KUKA KRL program: MyProgram_078().src

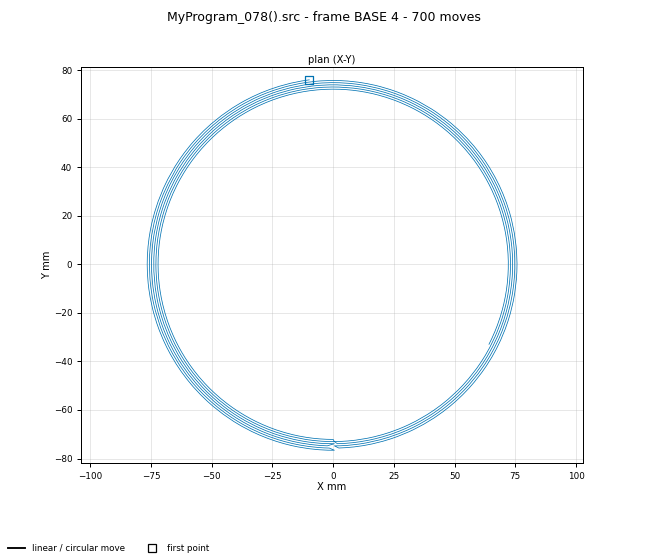
[picture p0: tool path of MyProgram_078().src in frame BASE 4, 700 of 700 moves have a stored position in this frame; points joined in program order, loops and branches not executed]
&ACCESS RVP
&REL 1
&PARAM TEMPLATE = C:\KRC\Roboter\Template\vorgabe
&PARAM EDITMASK = *
DEF MyProgram_078()
; ---- Setting reference (Base) ----
$BASE = BASE_DATA[4]

; --------------------------
; ---- Setting tool (TCP) ----
$TOOL = TOOL_DATA[3]
; --------------------------

$VEL.CP = VEL_APROX_PRINT
Startdeposition()
$VEL.CP = VEL_PRINT
LIN {X -9.8777,Y 75.9494,Z 80,A 92.1088,B 24.884,C -2.486,E1 24.9779,E2 -7.6791} C_DIS
LIN {X -13.075,Y 75.4658,Z 80,A 94.5265,B 24.8842,C -2.4842,E1 24.9713,E2 -10.0948} C_DIS
LIN {X -17.5111,Y 74.5607,Z 80,A 97.8703,B 24.8845,C -2.4802,E1 24.9622,E2 -13.4331} C_DIS
LIN {X -22.3044,Y 73.2687,Z 80,A 101.5575,B 24.885,C -2.4756,E1 24.9523,E2 -17.1153} C_DIS
LIN {X -26.0377,Y 72.0267,Z 80,A 104.8313,B 24.8845,C -2.4806,E1 24.9436,E2 -20.4073} C_DIS
LIN {X -29.6521,Y 70.616,Z 80,A 107.6677,B 24.885,C -2.4749,E1 24.9363,E2 -23.2364} C_DIS
LIN {X -33.18,Y 69.0287,Z 80,A 110.4546,B 24.8857,C -2.4677,E1 24.9292,E2 -26.0132} C_DIS
LIN {X -36.3303,Y 67.4239,Z 80,A 112.8541,B 24.8867,C -2.4571,E1 24.9233,E2 -28.394} C_DIS
LIN {X -38.0419,Y 66.4734,Z 80,A 114.6868,B 24.8861,C -2.4639,E1 24.9188,E2 -30.2484} C_DIS
LIN {X -41.522,Y 64.3565,Z 80,A 117.6505,B 24.8868,C -2.4562,E1 24.9118,E2 -33.2029} C_DIS
LIN {X -46.0253,Y 61.2172,Z 80,A 121.6077,B 24.8879,C -2.4442,E1 24.9029,E2 -37.1451} C_DIS
LIN {X -50.3353,Y 57.7255,Z 80,A 125.8636,B 24.8885,C -2.4378,E1 24.8937,E2 -41.402} C_DIS
LIN {X -53.3197,Y 54.9798,Z 80,A 129.0741,B 24.8887,C -2.4351,E1 24.8872,E2 -44.6194} C_DIS
LIN {X -56.3129,Y 51.9102,Z 80,A 132.6551,B 24.8886,C -2.4366,E1 24.8803,E2 -48.2195} C_DIS
LIN {X -58.7676,Y 49.1151,Z 80,A 135.4497,B 24.8892,C -2.4298,E1 24.8752,E2 -51.0105} C_DIS
LIN {X -61.2757,Y 45.9475,Z 80,A 137.8294,B 24.8914,C -2.4059,E1 24.8713,E2 -53.3446} C_DIS
LIN {X -63.0193,Y 43.5258,Z 80,A 140.4069,B 24.8912,C -2.4083,E1 24.8671,E2 -55.9405} C_DIS
LIN {X -65.1286,Y 40.3019,Z 80,A 143.5889,B 24.8912,C -2.4076,E1 24.8623,E2 -59.1371} C_DIS
LIN {X -68.074,Y 35.0981,Z 80,A 148.6418,B 24.8911,C -2.409,E1 24.8556,E2 -64.22} C_DIS
LIN {X -69.9567,Y 31.1775,Z 80,A 151.3838,B 24.8931,C -2.3867,E1 24.8525,E2 -66.9237} C_DIS
LIN {X -72.0828,Y 25.8816,Z 80,A 155.1336,B 24.8954,C -2.3611,E1 24.8488,E2 -70.6334} C_DIS
LIN {X -73.5664,Y 21.3077,Z 80,A 158.7364,B 24.8964,C -2.3501,E1 24.8458,E2 -74.2305} C_DIS
LIN {X -74.6505,Y 17.1227,Z 80,A 161.6509,B 24.8979,C -2.3323,E1 24.8438,E2 -77.1195} C_DIS
LIN {X -75.2853,Y 14.0748,Z 80,A 164.5038,B 24.8975,C -2.3375,E1 24.8422,E2 -80.0017} C_DIS
LIN {X -75.8096,Y 10.8996,Z 80,A 167.5902,B 24.8967,C -2.3464,E1 24.8409,E2 -83.1278} C_DIS
LIN {X -76.2313,Y 7.3889,Z 80,A 169.9673,B 24.898,C -2.3314,E1 24.8403,E2 -85.4835} C_DIS
LIN {X -76.5241,Y 3.1545,Z 80,A 172.7585,B 24.8997,C -2.312,E1 24.8399,E2 -88.2449} C_DIS
LIN {X -76.5895,Y -0.0837,Z 80,A 175.8098,B 24.8991,C -2.3195,E1 24.8399,E2 -91.3327} C_DIS
LIN {X -76.5051,Y -3.5969,Z 80,A 178.792,B 24.8991,C -2.3199,E1 24.8402,E2 -94.3338} C_DIS
LIN {X -76.1873,Y -7.835,Z 80,A -178.9442,B 24.9018,C -2.2875,E1 24.8408,E2 -96.5338} C_DIS
LIN {X -75.9118,Y -10.1663,Z 80,A -177.0242,B 24.902,C -2.286,E1 24.8415,E2 -98.4617} C_DIS
LIN {X -75.3667,Y -13.6289,Z 80,A -174.4282,B 24.9027,C -2.2773,E1 24.8427,E2 -101.0521} C_DIS
LIN {X -74.423,Y -18.0851,Z 80,A -171.3541,B 24.9043,C -2.2587,E1 24.8446,E2 -104.1} C_DIS
LIN {X -73.9363,Y -19.982,Z 80,A -168.6792,B 24.9021,C -2.284,E1 24.8466,E2 -106.851} C_DIS
LIN {X -72.7026,Y -24.0858,Z 80,A -166.4076,B 24.9049,C -2.2515,E1 24.8485,E2 -109.0578} C_DIS
LIN {X -71.6262,Y -27.1213,Z 80,A -164.2828,B 24.9061,C -2.2375,E1 24.8505,E2 -111.1612} C_DIS
LIN {X -69.8982,Y -31.3073,Z 80,A -160.4907,B 24.9061,C -2.2378,E1 24.8547,E2 -114.9751} C_DIS
LIN {X -68.5056,Y -34.2481,Z 80,A -157.5374,B 24.9055,C -2.244,E1 24.8584,E2 -117.959} C_DIS
LIN {X -66.9906,Y -37.1241,Z 80,A -155.5564,B 24.907,C -2.2262,E1 24.861,E2 -119.9081} C_DIS
LIN {X -64.6632,Y -41.045,Z 80,A -152.4733,B 24.9085,C -2.2091,E1 24.8654,E2 -122.9663} C_DIS
LIN {X -62.5538,Y -44.1917,Z 80,A -149.0219,B 24.9078,C -2.2175,E1 24.8709,E2 -126.4549} C_DIS
LIN {X -59.9723,Y -47.6364,Z 80,A -146.377,B 24.9096,C -2.1954,E1 24.8754,E2 -129.0594} C_DIS
LIN {X -57.6547,Y -50.4164,Z 80,A -143.0708,B 24.9089,C -2.2043,E1 24.8814,E2 -132.4021} C_DIS
LIN {X -54.7215,Y -53.5864,Z 80,A -140.3193,B 24.9104,C -2.1852,E1 24.8866,E2 -135.1198} C_DIS
LIN {X -51.7395,Y -56.4703,Z 80,A -137.0365,B 24.9106,C -2.1835,E1 24.8933,E2 -138.4121} C_DIS
LIN {X -49.3216,Y -58.5956,Z 80,A -134.2933,B 24.9102,C -2.1875,E1 24.8992,E2 -141.1756} C_DIS
LIN {X -45.3584,Y -61.713,Z 80,A -130.7861,B 24.9113,C -2.174,E1 24.9069,E2 -144.6634} C_DIS
LIN {X -40.9195,Y -64.7428,Z 80,A -126.5969,B 24.9115,C -2.1721,E1 24.9167,E2 -148.8618} C_DIS
LIN {X -37.7326,Y -66.6508,Z 80,A -123.7962,B 24.9118,C -2.1688,E1 24.9235,E2 -151.663} C_DIS
LIN {X -33.5371,Y -68.8558,Z 80,A -120.4898,B 24.9126,C -2.1581,E1 24.9317,E2 -154.9528} C_DIS
LIN {X -30.2404,Y -70.3655,Z 80,A -117.2499,B 24.9117,C -2.1693,E1 24.94,E2 -158.2269} C_DIS
LIN {X -26.7617,Y -71.7607,Z 80,A -114.3188,B 24.9117,C -2.1702,E1 24.9477,E2 -161.1663} C_DIS
LIN {X -23.5205,Y -72.888,Z 80,A -112.3294,B 24.9131,C -2.1525,E1 24.9529,E2 -163.1173} C_DIS
LIN {X -20.3575,Y -73.8336,Z 80,A -110.3071,B 24.9142,C -2.1388,E1 24.9582,E2 -165.1103} C_DIS
LIN {X -17.2131,Y -74.6297,Z 80,A -107.234,B 24.9129,C -2.155,E1 24.9667,E2 -168.2263} C_DIS
LIN {X -14.541,Y -75.196,Z 80,A -105.0876,B 24.9127,C -2.1571,E1 24.9726,E2 -170.38} C_DIS
LIN {X -9.9621,Y -75.9385,Z 80,A -101.7452,B 24.9131,C -2.1527,E1 24.9818,E2 -173.7147} C_DIS
LIN {X -5.8541,Y -76.3646,Z 80,A -99.0526,B 24.914,C -2.1415,E1 24.9892,E2 -176.3821} C_DIS
LIN {X -2.2483,Y -76.5559,Z 80,A -96.0072,B 24.9132,C -2.1514,E1 24.9978,E2 -179.4515} C_DIS
LIN {X 0.483,Y -76.5778,Z 80,A -94.1805,B 24.9136,C -2.1459,E1 25.0028,E2 -181.2653} C_DIS
Enddeposition()
LIN {X 0.483,Y -76.5778,Z 80,A -94.1805,B 24.9136,C -2.1459,E1 25.0028,E2 -181.2653} C_DIS
Startdeposition()
$VEL.CP = VEL_PRINT
LIN {X -1.5771,Y -75.6785,Z 80,A -96.5884,B 24.9143,C -2.1375,E1 24.9961,E2 -178.8375} C_DIS
LIN {X -3.5938,Y -75.6104,Z 80,A -98.116,B 24.9143,C -2.1374,E1 24.9918,E2 -177.3091} C_DIS
LIN {X -5.9465,Y -75.4611,Z 80,A -100.5202,B 24.9156,C -2.1208,E1 24.985,E2 -174.8646} C_DIS
LIN {X -10.1334,Y -75.0142,Z 80,A -103.377,B 24.9149,C -2.13,E1 24.9771,E2 -172.0279} C_DIS
LIN {X -13.7763,Y -74.4317,Z 80,A -105.7979,B 24.914,C -2.1407,E1 24.9705,E2 -169.6301} C_DIS
LIN {X -16.8855,Y -73.7877,Z 80,A -109.1458,B 24.9159,C -2.117,E1 24.9612,E2 -166.2216} C_DIS
LIN {X -20.0524,Y -72.9904,Z 80,A -110.7334,B 24.914,C -2.1416,E1 24.9571,E2 -164.69} C_DIS
LIN {X -22.5615,Y -72.2546,Z 80,A -113.5108,B 24.9155,C -2.1222,E1 24.9495,E2 -161.8618} C_DIS
LIN {X -26.4354,Y -70.9282,Z 80,A -116.6648,B 24.9155,C -2.1236,E1 24.9413,E2 -158.7046} C_DIS
LIN {X -29.9531,Y -69.5158,Z 80,A -119.1811,B 24.9145,C -2.1355,E1 24.9348,E2 -156.211} C_DIS
LIN {X -33.8293,Y -67.7146,Z 80,A -122.3374,B 24.914,C -2.1413,E1 24.9269,E2 -153.0603} C_DIS
LIN {X -37.0718,Y -65.9958,Z 80,A -124.7734,B 24.913,C -2.1537,E1 24.921,E2 -150.6469} C_DIS
LIN {X -39.3179,Y -64.6825,Z 80,A -126.8229,B 24.913,C -2.1544,E1 24.9161,E2 -148.593} C_DIS
LIN {X -41.771,Y -63.1263,Z 80,A -129.0307,B 24.9127,C -2.1576,E1 24.9109,E2 -146.3856} C_DIS
LIN {X -44.0945,Y -61.5258,Z 80,A -131.5383,B 24.9132,C -2.1518,E1 24.9051,E2 -143.8555} C_DIS
LIN {X -47.2138,Y -59.1659,Z 80,A -134.6288,B 24.913,C -2.1538,E1 24.8983,E2 -140.7585} C_DIS
LIN {X -50.1177,Y -56.7278,Z 80,A -137.766,B 24.913,C -2.1528,E1 24.8917,E2 -137.6065} C_DIS
LIN {X -53.6914,Y -53.3574,Z 80,A -140.5466,B 24.9106,C -2.1834,E1 24.8862,E2 -134.8874} C_DIS
LIN {X -55.2117,Y -51.7823,Z 80,A -143.3806,B 24.9126,C -2.1583,E1 24.8806,E2 -131.9811} C_DIS
LIN {X -57.7162,Y -48.9745,Z 80,A -145.892,B 24.9114,C -2.1729,E1 24.8761,E2 -129.493} C_DIS
LIN {X -60.2464,Y -45.8274,Z 80,A -148.8534,B 24.9107,C -2.1824,E1 24.8711,E2 -126.5403} C_DIS
LIN {X -63.1999,Y -41.6594,Z 80,A -152.3928,B 24.9092,C -2.1999,E1 24.8655,E2 -123.0252} C_DIS
LIN {X -65.9338,Y -37.1827,Z 80,A -156.1071,B 24.9078,C -2.2164,E1 24.8602,E2 -119.3312} C_DIS
LIN {X -67.8397,Y -33.5776,Z 80,A -159.079,B 24.9069,C -2.2276,E1 24.8564,E2 -116.37} C_DIS
LIN {X -70.1032,Y -28.5527,Z 80,A -163.5729,B 24.9066,C -2.2316,E1 24.8512,E2 -111.8611} C_DIS
LIN {X -71.1408,Y -25.8597,Z 80,A -166.1416,B 24.9068,C -2.2289,E1 24.8487,E2 -109.2714} C_DIS
LIN {X -73.3129,Y -18.84,Z 80,A -171.1553,B 24.9043,C -2.2584,E1 24.8447,E2 -104.2993} C_DIS
LIN {X -74.0337,Y -15.7716,Z 80,A -173.7321,B 24.9041,C -2.2611,E1 24.8431,E2 -101.7139} C_DIS
LIN {X -74.4465,Y -13.6945,Z 80,A -175.7304,B 24.9045,C -2.2568,E1 24.8421,E2 -99.6934} C_DIS
LIN {X -75.1155,Y -9.3522,Z 80,A -178.5608,B 24.9026,C -2.2788,E1 24.8409,E2 -96.8986} C_DIS
LIN {X -75.4572,Y -5.9942,Z 80,A 178.1742,B 24.9033,C -2.2702,E1 24.8401,E2 -93.5936} C_DIS
LIN {X -75.6918,Y 0.7374,Z 80,A 173.3776,B 24.9013,C -2.2934,E1 24.8398,E2 -88.8234} C_DIS
LIN {X -75.5872,Y 4.0345,Z 80,A 170.7099,B 24.901,C -2.2974,E1 24.8401,E2 -86.1493} C_DIS
LIN {X -75.3206,Y 7.5167,Z 80,A 168.0857,B 24.9002,C -2.3063,E1 24.8408,E2 -83.5305} C_DIS
LIN {X -74.7463,Y 11.9525,Z 80,A 165.1359,B 24.8984,C -2.3271,E1 24.8419,E2 -80.6129} C_DIS
LIN {X -73.7542,Y 17.0307,Z 80,A 160.4984,B 24.8988,C -2.3227,E1 24.8446,E2 -75.9375} C_DIS
LIN {X -72.6569,Y 21.2318,Z 80,A 156.66,B 24.899,C -2.3203,E1 24.8475,E2 -72.071} C_DIS
LIN {X -71.4063,Y 25.117,Z 80,A 154.6372,B 24.896,C -2.3544,E1 24.8493,E2 -70.1183} C_DIS
LIN {X -70.0146,Y 28.7687,Z 80,A 151.3832,B 24.8958,C -2.3565,E1 24.8526,E2 -66.851} C_DIS
LIN {X -68.1089,Y 32.9209,Z 80,A 148.5531,B 24.8935,C -2.3823,E1 24.8558,E2 -64.0671} C_DIS
LIN {X -64.5667,Y 39.5085,Z 80,A 142.8168,B 24.8923,C -2.3961,E1 24.8635,E2 -58.3334} C_DIS
LIN {X -62.8936,Y 42.1203,Z 80,A 139.9656,B 24.8927,C -2.3907,E1 24.8678,E2 -55.4549} C_DIS
LIN {X -61.2571,Y 44.4679,Z 80,A 137.5513,B 24.8927,C -2.3907,E1 24.8718,E2 -53.0287} C_DIS
LIN {X -58.5287,Y 48.0021,Z 80,A 134.3381,B 24.8916,C -2.4034,E1 24.8773,E2 -49.8309} C_DIS
LIN {X -55.7959,Y 51.1522,Z 80,A 131.0027,B 24.8913,C -2.4071,E1 24.8835,E2 -46.4893} C_DIS
LIN {X -52.8118,Y 54.2265,Z 80,A 127.5163,B 24.8911,C -2.4091,E1 24.8904,E2 -42.9928} C_DIS
LIN {X -50.1761,Y 56.6759,Z 80,A 124.7811,B 24.8906,C -2.4149,E1 24.8961,E2 -40.2606} C_DIS
LIN {X -46.3964,Y 59.8094,Z 80,A 121.4177,B 24.8891,C -2.4314,E1 24.9034,E2 -36.924} C_DIS
LIN {X -43.5152,Y 61.9371,Z 80,A 119.0724,B 24.8877,C -2.4458,E1 24.9086,E2 -34.6049} C_DIS
LIN {X -39.3079,Y 64.6885,Z 80,A 114.706,B 24.8883,C -2.4392,E1 24.9189,E2 -30.2086} C_DIS
LIN {X -36.5712,Y 66.2751,Z 80,A 112.1957,B 24.8883,C -2.4405,E1 24.925,E2 -27.6941} C_DIS
LIN {X -32.5759,Y 68.3271,Z 80,A 109.1203,B 24.887,C -2.4539,E1 24.9327,E2 -24.6426} C_DIS
LIN {X -29.8634,Y 69.5545,Z 80,A 106.9712,B 24.8864,C -2.4598,E1 24.9381,E2 -22.5024} C_DIS
LIN {X -27.5483,Y 70.5041,Z 80,A 104.5385,B 24.8874,C -2.4489,E1 24.9445,E2 -20.0384} C_DIS
LIN {X -24.5534,Y 71.6031,Z 80,A 102.4647,B 24.8864,C -2.4604,E1 24.9499,E2 -17.9879} C_DIS
LIN {X -20.0121,Y 73.0011,Z 80,A 98.9131,B 24.8859,C -2.4655,E1 24.9594,E2 -14.4425} C_DIS
LIN {X -18.0186,Y 73.5191,Z 80,A 96.4429,B 24.8879,C -2.4439,E1 24.9663,E2 -11.9177} C_DIS
LIN {X -14.0327,Y 74.3834,Z 80,A 94.194,B 24.8857,C -2.4677,E1 24.9723,E2 -9.7227} C_DIS
LIN {X -10.9409,Y 74.9005,Z 80,A 91.886,B 24.8854,C -2.4709,E1 24.9786,E2 -7.4204} C_DIS
LIN {X -7.0765,Y 75.3635,Z 80,A 89.3928,B 24.8842,C -2.4843,E1 24.9855,E2 -4.9575} C_DIS
LIN {X -5.0644,Y 75.5253,Z 80,A 86.3304,B 24.8878,C -2.4453,E1 24.9943,E2 -1.8011} C_DIS
LIN {X -0.5418,Y 75.6931,Z 80,A 83.9367,B 24.8852,C -2.4728,E1 25.0008,E2 0.5272} C_DIS
LIN {X 2.7502,Y 75.6446,Z 80,A 80.8301,B 24.8867,C -2.457,E1 25.0096,E2 3.6708} C_DIS
LIN {X 6.086,Y 75.4495,Z 80,A 78.59,B 24.886,C -2.4645,E1 25.0157,E2 5.8921} C_DIS
LIN {X 10.3575,Y 74.9835,Z 80,A 75.5916,B 24.8854,C -2.4705,E1 25.024,E2 8.8737} C_DIS
LIN {X 13.8407,Y 74.4196,Z 80,A 72.3601,B 24.8869,C -2.4546,E1 25.033,E2 12.1395} C_DIS
LIN {X 17.1405,Y 73.7288,Z 80,A 70.7874,B 24.8846,C -2.4797,E1 25.0371,E2 13.6506} C_DIS
LIN {X 19.3068,Y 73.1924,Z 80,A 68.1739,B 24.887,C -2.4536,E1 25.0443,E2 16.3218} C_DIS
LIN {X 23.3915,Y 71.9901,Z 80,A 64.9215,B 24.8873,C -2.4503,E1 25.053,E2 19.576} C_DIS
LIN {X 26.5408,Y 70.8889,Z 80,A 63.1766,B 24.8856,C -2.4693,E1 25.0574,E2 21.2722} C_DIS
LIN {X 29.0873,Y 69.8825,Z 80,A 60.9184,B 24.8862,C -2.4621,E1 25.0633,E2 23.5423} C_DIS
LIN {X 32.7666,Y 68.2354,Z 80,A 57.806,B 24.8867,C -2.4569,E1 25.0712,E2 26.6592} C_DIS
LIN {X 35.2397,Y 66.9914,Z 80,A 55.4646,B 24.8876,C -2.4474,E1 25.077,E2 29.0166} C_DIS
LIN {X 40.4766,Y 63.9653,Z 80,A 51.5107,B 24.8866,C -2.4582,E1 25.0864,E2 32.9328} C_DIS
LIN {X 42.3299,Y 62.7522,Z 80,A 49.2882,B 24.8882,C -2.4402,E1 25.0917,E2 35.1905} C_DIS
LIN {X 46.4154,Y 59.7947,Z 80,A 45.9821,B 24.8875,C -2.448,E1 25.099,E2 38.4663} C_DIS
LIN {X 48.6468,Y 57.9943,Z 80,A 43.5524,B 24.8886,C -2.4366,E1 25.1043,E2 40.9138} C_DIS
LIN {X 51.5182,Y 55.46,Z 80,A 40.6828,B 24.889,C -2.4317,E1 25.1102,E2 43.7835} C_DIS
LIN {X 55.0143,Y 51.9922,Z 80,A 36.9651,B 24.8897,C -2.4241,E1 25.1175,E2 47.5033} C_DIS
LIN {X 57.9548,Y 48.6943,Z 80,A 33.8949,B 24.8897,C -2.4244,E1 25.1232,E2 50.5588} C_DIS
LIN {X 60.4112,Y 45.6097,Z 80,A 30.3734,B 24.8917,C -2.4018,E1 25.1293,E2 54.1173} C_DIS
LIN {X 62.6825,Y 42.4339,Z 80,A 27.2188,B 24.8929,C -2.3886,E1 25.1343,E2 57.2876} C_DIS
LIN {X 64.457,Y 39.6885,Z 80,A 24.8099,B 24.8933,C -2.384,E1 25.1378,E2 59.695} C_DIS
LIN {X 66.5079,Y 36.1446,Z 80,A 22.251,B 24.8927,C -2.3916,E1 25.1412,E2 62.2227} C_DIS
LIN {X 68.5159,Y 32.1771,Z 80,A 18.8456,B 24.8936,C -2.3811,E1 25.1455,E2 65.6347} C_DIS
LIN {X 69.8894,Y 29.0708,Z 80,A 15.5268,B 24.8962,C -2.3518,E1 25.1491,E2 69.0043} C_DIS
LIN {X 71.3051,Y 25.4018,Z 80,A 13.913,B 24.8934,C -2.3834,E1 25.1506,E2 70.5345} C_DIS
LIN {X 72.6316,Y 21.3171,Z 80,A 10.1653,B 24.8956,C -2.3589,E1 25.1538,E2 74.3188} C_DIS
LIN {X 73.3917,Y 18.5285,Z 80,A 7.457,B 24.8975,C -2.3369,E1 25.1557,E2 77.0636} C_DIS
LIN {X 74.604,Y 12.8095,Z 80,A 3.9207,B 24.8964,C -2.3497,E1 25.1576,E2 80.5489} C_DIS
LIN {X 75.3352,Y 7.3665,Z 80,A -0.1483,B 24.8973,C -2.3394,E1 25.1591,E2 84.6184} C_DIS
LIN {X 75.5228,Y 5.1018,Z 80,A -2.2389,B 24.8988,C -2.3228,E1 25.1595,E2 86.7356} C_DIS
LIN {X 75.694,Y 0.335,Z 80,A -6.1723,B 24.9006,C -2.3017,E1 25.1598,E2 90.6955} C_DIS
LIN {X 75.6309,Y -3.1149,Z 80,A -8.384,B 24.9003,C -2.3054,E1 25.1596,E2 92.8855} C_DIS
LIN {X 75.4373,Y -6.2402,Z 80,A -10.8516,B 24.9012,C -2.2949,E1 25.1591,E2 95.3632} C_DIS
LIN {X 74.7333,Y -12.0356,Z 80,A -14.9146,B 24.9015,C -2.2915,E1 25.1576,E2 99.4102} C_DIS
LIN {X 74.1249,Y -15.3364,Z 80,A -17.626,B 24.9026,C -2.2783,E1 25.1562,E2 102.1368} C_DIS
LIN {X 72.95,Y -20.198,Z 80,A -21.0846,B 24.9028,C -2.2763,E1 25.1539,E2 105.5803} C_DIS
LIN {X 71.9928,Y -23.3813,Z 80,A -24.6347,B 24.9061,C -2.2376,E1 25.1508,E2 109.2016} C_DIS
LIN {X 70.8117,Y -26.7476,Z 80,A -26.1131,B 24.9037,C -2.2658,E1 25.1495,E2 110.605} C_DIS
LIN {X 68.9544,Y -31.2255,Z 80,A -30.6307,B 24.9068,C -2.2293,E1 25.1445,E2 115.184} C_DIS
LIN {X 67.1287,Y -34.9777,Z 80,A -33.3836,B 24.9065,C -2.2321,E1 25.1411,E2 117.9157} C_DIS
LIN {X 65.3574,Y -38.1859,Z 80,A -36.6198,B 24.9083,C -2.2104,E1 25.1365,E2 121.1864} C_DIS
LIN {X 63.124,Y -41.7745,Z 80,A -40.0037,B 24.9095,C -2.1961,E1 25.1314,E2 124.5873} C_DIS
LIN {X 61.155,Y -44.6072,Z 80,A -41.8497,B 24.9083,C -2.2115,E1 25.1284,E2 126.3878} C_DIS
LIN {X 58.0862,Y -48.5361,Z 80,A -45.7317,B 24.9093,C -2.1984,E1 25.1216,E2 130.2827} C_DIS
LIN {X 55.8549,Y -51.0879,Z 80,A -48.965,B 24.9115,C -2.1724,E1 25.1155,E2 133.563} C_DIS
LIN {X 53.3412,Y -53.7074,Z 80,A -50.9656,B 24.9102,C -2.1876,E1 25.1117,E2 135.5193} C_DIS
LIN {X 50.6173,Y -56.2818,Z 80,A -53.7997,B 24.9108,C -2.181,E1 25.1058,E2 138.3573} C_DIS
LIN {X 48.1407,Y -58.4149,Z 80,A -56.5393,B 24.9119,C -2.1678,E1 25.0999,E2 141.1176} C_DIS
LIN {X 45.1335,Y -60.7689,Z 80,A -59.3124,B 24.9121,C -2.1651,E1 25.0938,E2 143.8869} C_DIS
LIN {X 41.5011,Y -63.3042,Z 80,A -62.0188,B 24.9111,C -2.1772,E1 25.0876,E2 146.5557} C_DIS
LIN {X 37.2963,Y -65.8691,Z 80,A -66.1577,B 24.9126,C -2.1585,E1 25.0777,E2 150.7259} C_DIS
LIN {X 32.9711,Y -68.1372,Z 80,A -69.461,B 24.9122,C -2.1636,E1 25.0695,E2 154.008} C_DIS
LIN {X 31.1012,Y -69.0104,Z 80,A -72.6307,B 24.916,C -2.1159,E1 25.0612,E2 157.2829} C_DIS
LIN {X 26.5262,Y -70.8944,Z 80,A -74.8606,B 24.913,C -2.1533,E1 25.0556,E2 159.4193} C_DIS
LIN {X 23.8179,Y -71.8495,Z 80,A -77.9876,B 24.9154,C -2.1238,E1 25.0472,E2 162.6099} C_DIS
LIN {X 20.5212,Y -72.8601,Z 80,A -79.7557,B 24.9138,C -2.1444,E1 25.0426,E2 164.3263} C_DIS
LIN {X 15.9944,Y -73.986,Z 80,A -83.4595,B 24.9144,C -2.1362,E1 25.0325,E2 168.0444} C_DIS
LIN {X 12.3827,Y -74.6753,Z 80,A -86.266,B 24.9146,C -2.1333,E1 25.0247,E2 170.8545} C_DIS
LIN {X 8.6061,Y -75.204,Z 80,A -89.1905,B 24.9149,C -2.1304,E1 25.0166,E2 173.7835} C_DIS
LIN {X 5.4445,Y -75.4989,Z 80,A -91.5056,B 24.9148,C -2.1317,E1 25.0102,E2 176.0944} C_DIS
LIN {X 2.3291,Y -75.6591,Z 80,A -94.7094,B 24.9167,C -2.1081,E1 25.0011,E2 179.3533} C_DIS
LIN {X 2.3291,Y -75.6591,Z 80,A -94.7094,B 24.9167,C -2.1081,E1 25.0011,E2 179.3533} C_DIS
Enddeposition()
LIN {X 0.4812,Y -74.7699,Z 80,A -95.2576,B 24.9136,C -2.1469,E1 24.9998,E2 179.8095} C_DIS
Startdeposition()
$VEL.CP = VEL_PRINT
LIN {X 2.812,Y -74.7476,Z 80,A -92.4237,B 24.9112,C -2.1753,E1 25.0079,E2 176.9086} C_DIS
LIN {X 5.9383,Y -74.5647,Z 80,A -90.0902,B 24.9113,C -2.1746,E1 25.0144,E2 174.5779} C_DIS
LIN {X 10.5837,Y -74.0484,Z 80,A -86.7702,B 24.9117,C -2.1695,E1 25.0236,E2 171.2724} C_DIS
LIN {X 13.6044,Y -73.554,Z 80,A -83.8358,B 24.9102,C -2.1877,E1 25.0318,E2 168.2979} C_DIS
LIN {X 19.3007,Y -72.2683,Z 80,A -79.7389,B 24.9107,C -2.1814,E1 25.0429,E2 164.2217} C_DIS
LIN {X 22.9194,Y -71.2032,Z 80,A -76.547,B 24.9098,C -2.1933,E1 25.0514,E2 161.0074} C_DIS
LIN {X 26.8746,Y -69.8074,Z 80,A -72.7517,B 24.908,C -2.2143,E1 25.0615,E2 157.1706} C_DIS
LIN {X 30.3396,Y -68.3725,Z 80,A -70.6516,B 24.9095,C -2.1963,E1 25.0667,E2 155.1181} C_DIS
LIN {X 33.2038,Y -67.0272,Z 80,A -68.3254,B 24.9095,C -2.1973,E1 25.0725,E2 152.7955} C_DIS
LIN {X 35.4029,Y -65.8928,Z 80,A -66.0422,B 24.9082,C -2.2118,E1 25.0782,E2 150.4847} C_DIS
LIN {X 39.9804,Y -63.2212,Z 80,A -61.7012,B 24.9069,C -2.2275,E1 25.0886,E2 146.1201} C_DIS
LIN {X 42.6642,Y -61.4397,Z 80,A -59.6412,B 24.9075,C -2.2205,E1 25.0933,E2 144.0838} C_DIS
LIN {X 45.9769,Y -59.0017,Z 80,A -56.4694,B 24.9069,C -2.2277,E1 25.1004,E2 140.9063} C_DIS
LIN {X 48.3902,Y -57.0403,Z 80,A -54.4365,B 24.9073,C -2.2227,E1 25.1047,E2 138.8931} C_DIS
LIN {X 51.4102,Y -54.333,Z 80,A -51.2033,B 24.9064,C -2.2336,E1 25.1114,E2 135.6471} C_DIS
LIN {X 54.0361,Y -51.7229,Z 80,A -48.1986,B 24.9054,C -2.2455,E1 25.1173,E2 132.6272} C_DIS
LIN {X 55.8891,Y -49.7155,Z 80,A -46.3181,B 24.9054,C -2.2445,E1 25.1208,E2 130.7575} C_DIS
LIN {X 59.7471,Y -45.0051,Z 80,A -42.0825,B 24.9055,C -2.2439,E1 25.1282,E2 126.5429} C_DIS
LIN {X 62.6709,Y -40.8362,Z 80,A -38.2243,B 24.9047,C -2.2533,E1 25.1343,E2 122.6814} C_DIS
LIN {X 64.4742,Y -37.9246,Z 80,A -34.9338,B 24.9024,C -2.2807,E1 25.1391,E2 119.343} C_DIS
LIN {X 66.2003,Y -34.8232,Z 80,A -32.7037,B 24.903,C -2.2739,E1 25.1421,E2 117.1407} C_DIS
LIN {X 68.0942,Y -30.9583,Z 80,A -29.6504,B 24.9028,C -2.2764,E1 25.1458,E2 114.0979} C_DIS
LIN {X 69.6296,Y -27.3294,Z 80,A -26.6007,B 24.9019,C -2.2864,E1 25.1491,E2 111.0413} C_DIS
LIN {X 71.6282,Y -21.5532,Z 80,A -22.1045,B 24.9012,C -2.2952,E1 25.1531,E2 106.5498} C_DIS
LIN {X 72.9563,Y -16.5124,Z 80,A -17.4227,B 24.8983,C -2.3284,E1 25.1564,E2 101.8164} C_DIS
LIN {X 73.8228,Y -12.0599,Z 80,A -13.4403,B 24.8959,C -2.3549,E1 25.1583,E2 97.7949} C_DIS
LIN {X 74.3269,Y -8.4086,Z 80,A -11.3147,B 24.897,C -2.3426,E1 25.159,E2 95.7107} C_DIS
LIN {X 74.6276,Y -5.0883,Z 80,A -8.8673,B 24.8966,C -2.3476,E1 25.1595,E2 93.2662} C_DIS
LIN {X 74.7805,Y -1.7516,Z 80,A -6.191,B 24.8956,C -2.3593,E1 25.1598,E2 90.5781} C_DIS
LIN {X 74.7622,Y 2.409,Z 80,A -3.4856,B 24.8959,C -2.3549,E1 25.1597,E2 87.8992} C_DIS
LIN {X 74.6559,Y 4.6529,Z 80,A -1.4171,B 24.8945,C -2.3708,E1 25.1593,E2 85.8055} C_DIS
LIN {X 74.3647,Y 8.0611,Z 80,A 1.4492,B 24.8931,C -2.3865,E1 25.1586,E2 82.9191} C_DIS
LIN {X 73.8505,Y 11.8943,Z 80,A 4.7657,B 24.8913,C -2.4064,E1 25.1571,E2 79.5751} C_DIS
LIN {X 73.2334,Y 15.234,Z 80,A 6.7132,B 24.8924,C -2.3946,E1 25.1561,E2 77.6667} C_DIS
LIN {X 72.3845,Y 18.8602,Z 80,A 9.5137,B 24.8918,C -2.4017,E1 25.1542,E2 74.8657} C_DIS
LIN {X 71.1715,Y 23.0171,Z 80,A 13.0341,B 24.8903,C -2.4177,E1 25.1513,E2 71.3275} C_DIS
LIN {X 70.3093,Y 25.5299,Z 80,A 15.355,B 24.889,C -2.4322,E1 25.1491,E2 68.9853} C_DIS
LIN {X 68.6095,Y 29.7973,Z 80,A 18.2292,B 24.8898,C -2.423,E1 25.146,E2 66.1487} C_DIS
LIN {X 67.4211,Y 32.3971,Z 80,A 20.6833,B 24.8885,C -2.437,E1 25.1431,E2 63.6749} C_DIS
LIN {X 65.8164,Y 35.5442,Z 80,A 23.5357,B 24.8875,C -2.4487,E1 25.1393,E2 60.8099} C_DIS
LIN {X 62.8617,Y 40.5415,Z 80,A 27.6478,B 24.8873,C -2.4503,E1 25.1334,E2 56.7148} C_DIS
LIN {X 61.0178,Y 43.2672,Z 80,A 30.3791,B 24.8862,C -2.4628,E1 25.129,E2 53.9673} C_DIS
LIN {X 57.5907,Y 47.7335,Z 80,A 34.5261,B 24.8857,C -2.4681,E1 25.1218,E2 49.8271} C_DIS
LIN {X 55.1061,Y 50.5815,Z 80,A 37.3812,B 24.8852,C -2.4734,E1 25.1165,E2 46.9723} C_DIS
LIN {X 52.2671,Y 53.5111,Z 80,A 40.2054,B 24.8854,C -2.4713,E1 25.111,E2 44.165} C_DIS
LIN {X 50.4341,Y 55.2414,Z 80,A 42.3699,B 24.8844,C -2.482,E1 25.1065,E2 41.9841} C_DIS
LIN {X 47.4522,Y 57.8235,Z 80,A 45.3604,B 24.8839,C -2.4868,E1 25.1002,E2 38.9939} C_DIS
LIN {X 43.9521,Y 60.5252,Z 80,A 49.3052,B 24.8819,C -2.5087,E1 25.0913,E2 35.0113} C_DIS
LIN {X 41.2743,Y 62.3828,Z 80,A 51.1306,B 24.8833,C -2.4936,E1 25.0871,E2 33.2278} C_DIS
LIN {X 38.7436,Y 63.9853,Z 80,A 53.6081,B 24.8825,C -2.5022,E1 25.0812,E2 30.7378} C_DIS
LIN {X 34.533,Y 66.3524,Z 80,A 56.6845,B 24.8836,C -2.4897,E1 25.0738,E2 27.6998} C_DIS
LIN {X 30.9922,Y 68.0786,Z 80,A 60.2601,B 24.8818,C -2.5089,E1 25.0647,E2 24.0883} C_DIS
LIN {X 28.4244,Y 69.1899,Z 80,A 62.2462,B 24.882,C -2.5068,E1 25.0596,E2 22.1118} C_DIS
LIN {X 25.6595,Y 70.2621,Z 80,A 64.8765,B 24.8809,C -2.5188,E1 25.0527,E2 19.4586} C_DIS
LIN {X 22.5779,Y 71.3134,Z 80,A 67.4863,B 24.8804,C -2.5239,E1 25.0457,E2 16.8415} C_DIS
LIN {X 18.6435,Y 72.4403,Z 80,A 70.051,B 24.8817,C -2.5103,E1 25.0389,E2 14.3131} C_DIS
LIN {X 13.4747,Y 73.5776,Z 80,A 74.0849,B 24.8816,C -2.5116,E1 25.0279,E2 10.2813} C_DIS
LIN {X 9.8948,Y 74.1441,Z 80,A 76.9996,B 24.8812,C -2.5161,E1 25.0198,E2 7.3586} C_DIS
LIN {X 6.7902,Y 74.492,Z 80,A 80.3304,B 24.8787,C -2.5416,E1 25.0104,E2 3.9692} C_DIS
LIN {X 2.7304,Y 74.7507,Z 80,A 81.9274,B 24.8826,C -2.501,E1 25.0062,E2 2.4693} C_DIS
LIN {X -0.7522,Y 74.7977,Z 80,A 86.0605,B 24.879,C -2.5392,E1 24.9944,E2 -1.7545} C_DIS
LIN {X -4.6442,Y 74.6565,Z 80,A 87.9785,B 24.8817,C -2.51,E1 24.9893,E2 -3.6037} C_DIS
LIN {X -7.0504,Y 74.4677,Z 80,A 90.2171,B 24.8809,C -2.5193,E1 24.983,E2 -5.8655} C_DIS
LIN {X -12.028,Y 73.8281,Z 80,A 93.5546,B 24.8823,C -2.5038,E1 24.9738,E2 -9.1685} C_DIS
LIN {X -17.5464,Y 72.7132,Z 80,A 98.0526,B 24.8823,C -2.5049,E1 24.9615,E2 -13.6745} C_DIS
LIN {X -22.5224,Y 71.3306,Z 80,A 102.1544,B 24.8823,C -2.5043,E1 24.9505,E2 -17.7817} C_DIS
LIN {X -25.206,Y 70.4255,Z 80,A 104.4085,B 24.8823,C -2.5038,E1 24.9445,E2 -20.0389} C_DIS
LIN {X -30.0757,Y 68.4883,Z 80,A 108.2153,B 24.8833,C -2.493,E1 24.9347,E2 -23.8285} C_DIS
LIN {X -31.9713,Y 67.6247,Z 80,A 110.3235,B 24.8824,C -2.5034,E1 24.9293,E2 -25.9668} C_DIS
LIN {X -36.8142,Y 65.1156,Z 80,A 115.527,B 24.8806,C -2.5222,E1 24.9165,E2 -31.2299} C_DIS
LIN {X -41.2915,Y 62.3715,Z 80,A 118.1988,B 24.8845,C -2.4808,E1 24.9104,E2 -33.8118} C_DIS
LIN {X -43.7699,Y 60.6578,Z 80,A 120.8852,B 24.884,C -2.4855,E1 24.9043,E2 -36.5187} C_DIS
LIN {X -47.1298,Y 58.0858,Z 80,A 123.8792,B 24.8852,C -2.4726,E1 24.8977,E2 -39.4929} C_DIS
LIN {X -49.8558,Y 55.7635,Z 80,A 126.4368,B 24.8862,C -2.462,E1 24.8924,E2 -42.0352} C_DIS
LIN {X -52.6111,Y 53.1715,Z 80,A 129.4619,B 24.8866,C -2.4583,E1 24.8863,E2 -45.064} C_DIS
LIN {X -54.8474,Y 50.8623,Z 80,A 132.0749,B 24.8868,C -2.4559,E1 24.8813,E2 -47.6827} C_DIS
LIN {X -56.8541,Y 48.6087,Z 80,A 134.1595,B 24.8878,C -2.4446,E1 24.8775,E2 -49.7498} C_DIS
LIN {X -58.8273,Y 46.2013,Z 80,A 137.1462,B 24.8871,C -2.4529,E1 24.8722,E2 -52.7702} C_DIS
LIN {X -61.6496,Y 42.3614,Z 80,A 141.0011,B 24.8875,C -2.4479,E1 24.866,E2 -56.6322} C_DIS
LIN {X -63.5056,Y 39.525,Z 80,A 142.6669,B 24.8902,C -2.4184,E1 24.8636,E2 -58.2361} C_DIS
LIN {X -65.7928,Y 35.5878,Z 80,A 146.1256,B 24.8912,C -2.4078,E1 24.8588,E2 -61.6873} C_DIS
LIN {X -67.3861,Y 32.4686,Z 80,A 149.6171,B 24.8902,C -2.419,E1 24.8544,E2 -65.2245} C_DIS
LIN {X -68.9618,Y 28.9728,Z 80,A 152.1017,B 24.892,C -2.3995,E1 24.8517,E2 -67.6763} C_DIS
LIN {X -70.3827,Y 25.3252,Z 80,A 155.0202,B 24.8929,C -2.3885,E1 24.8488,E2 -70.5849} C_DIS
LIN {X -71.7019,Y 21.3076,Z 80,A 157.9073,B 24.8946,C -2.3703,E1 24.8464,E2 -73.4449} C_DIS
LIN {X -72.3095,Y 19.1479,Z 80,A 160.4146,B 24.8934,C -2.3834,E1 24.8445,E2 -75.9981} C_DIS
LIN {X -73.6522,Y 13.0597,Z 80,A 164.6723,B 24.8958,C -2.3562,E1 24.8421,E2 -80.2158} C_DIS
LIN {X -74.0363,Y 10.6684,Z 80,A 166.8589,B 24.8957,C -2.358,E1 24.8412,E2 -82.42} C_DIS
LIN {X -74.4094,Y 7.6447,Z 80,A 169.9649,B 24.8947,C -2.3689,E1 24.8403,E2 -85.5705} C_DIS
LIN {X -74.6993,Y 3.8963,Z 80,A 171.7319,B 24.8978,C -2.3335,E1 24.84,E2 -87.2636} C_DIS
LIN {X -74.7847,Y 1.567,Z 80,A 174.9828,B 24.8953,C -2.3624,E1 24.8398,E2 -90.6032} C_DIS
LIN {X -74.7377,Y -3.077,Z 80,A 178.3131,B 24.8968,C -2.3457,E1 24.8402,E2 -93.9136} C_DIS
LIN {X -74.4727,Y -6.9933,Z 80,A -179.5693,B 24.8994,C -2.3152,E1 24.8407,E2 -95.971} C_DIS
LIN {X -74.1982,Y -9.4773,Z 80,A -177.219,B 24.8991,C -2.3195,E1 24.8415,E2 -98.3457} C_DIS
LIN {X -73.487,Y -13.9596,Z 80,A -174.0912,B 24.9007,C -2.3005,E1 24.8429,E2 -101.4467} C_DIS
LIN {X -72.7573,Y -17.3636,Z 80,A -171.63,B 24.9018,C -2.2875,E1 24.8444,E2 -103.8913} C_DIS
LIN {X -72.1522,Y -19.7295,Z 80,A -168.6267,B 24.9,C -2.3089,E1 24.8467,E2 -106.9631} C_DIS
LIN {X -70.987,Y -23.5784,Z 80,A -166.3654,B 24.9025,C -2.2801,E1 24.8486,E2 -109.1687} C_DIS
LIN {X -69.8409,Y -26.7864,Z 80,A -162.8537,B 24.9012,C -2.2943,E1 24.8522,E2 -112.7339} C_DIS
LIN {X -68.2468,Y -30.6192,Z 80,A -160.6116,B 24.904,C -2.2627,E1 24.8546,E2 -114.9129} C_DIS
LIN {X -67.3815,Y -32.4796,Z 80,A -158.8585,B 24.904,C -2.2627,E1 24.8567,E2 -116.6756} C_DIS
LIN {X -65.6605,Y -35.8317,Z 80,A -156.077,B 24.9048,C -2.2523,E1 24.8603,E2 -119.4472} C_DIS
LIN {X -63.4924,Y -39.5462,Z 80,A -153.1744,B 24.9064,C -2.2343,E1 24.8644,E2 -122.3216} C_DIS
LIN {X -62.2009,Y -41.5492,Z 80,A -149.8361,B 24.9036,C -2.2666,E1 24.8698,E2 -125.7539} C_DIS
LIN {X -59.4863,Y -45.3503,Z 80,A -147.3668,B 24.9067,C -2.2306,E1 24.8738,E2 -128.1491} C_DIS
LIN {X -56.4128,Y -49.1201,Z 80,A -143.2097,B 24.9065,C -2.2327,E1 24.8813,E2 -132.3303} C_DIS
LIN {X -54.0506,Y -51.7084,Z 80,A -140.9106,B 24.9078,C -2.2174,E1 24.8856,E2 -134.6028} C_DIS
LIN {X -49.0215,Y -56.4989,Z 80,A -136.0706,B 24.9096,C -2.1947,E1 24.8954,E2 -139.4086} C_DIS
LIN {X -46.404,Y -58.6672,Z 80,A -132.4286,B 24.9079,C -2.216,E1 24.9034,E2 -143.115} C_DIS
LIN {X -42.642,Y -61.456,Z 80,A -129.3056,B 24.9094,C -2.1982,E1 24.9105,E2 -146.2065} C_DIS
LIN {X -39.8407,Y -63.3084,Z 80,A -126.5622,B 24.9094,C -2.1986,E1 24.9169,E2 -148.9597} C_DIS
LIN {X -37.0046,Y -65.0071,Z 80,A -124.1194,B 24.9098,C -2.1928,E1 24.9228,E2 -151.3959} C_DIS
LIN {X -34.124,Y -66.5637,Z 80,A -121.3393,B 24.9095,C -2.1966,E1 24.9297,E2 -154.1927} C_DIS
LIN {X -29.5386,Y -68.7209,Z 80,A -118.0855,B 24.9112,C -2.1761,E1 24.9379,E2 -157.4057} C_DIS
LIN {X -26.4411,Y -69.9718,Z 80,A -115.4907,B 24.9113,C -2.1745,E1 24.9446,E2 -160.0025} C_DIS
LIN {X -23.3032,Y -71.0779,Z 80,A -112.7172,B 24.911,C -2.1783,E1 24.952,E2 -162.7903} C_DIS
LIN {X -20.6856,Y -71.8843,Z 80,A -110.2462,B 24.9103,C -2.1867,E1 24.9587,E2 -165.2853} C_DIS
LIN {X -16.5579,Y -72.9458,Z 80,A -107.3413,B 24.9112,C -2.1755,E1 24.9665,E2 -168.1674} C_DIS
LIN {X -13.3052,Y -73.6081,Z 80,A -104.7319,B 24.9112,C -2.1763,E1 24.9737,E2 -170.7816} C_DIS
LIN {X -9.2495,Y -74.2272,Z 80,A -100.9193,B 24.9097,C -2.1938,E1 24.9844,E2 -174.6387} C_DIS
LIN {X -5.6937,Y -74.5835,Z 80,A -98.8673,B 24.9113,C -2.1751,E1 24.99,E2 -176.6471} C_DIS
LIN {X -2.4448,Y -74.7611,Z 80,A -95.3893,B 24.909,C -2.2024,E1 24.9998,E2 -180.1905} C_DIS
LIN {X -2.4448,Y -74.7611,Z 80,A -95.3893,B 24.909,C -2.2024,E1 24.9998,E2 -180.1905} C_DIS
Enddeposition()
LIN {X 0.4796,Y -73.8887,Z 80,A -95.0297,B 24.9119,C -2.1674,E1 25.0006,E2 -180.4671} C_DIS
Startdeposition()
$VEL.CP = VEL_PRINT
LIN {X -2.905,Y -73.8495,Z 80,A -97.9552,B 24.9126,C -2.1587,E1 24.9924,E2 -177.5207} C_DIS
LIN {X -5.7008,Y -73.6864,Z 80,A -101.1444,B 24.9147,C -2.1324,E1 24.9833,E2 -174.2677} C_DIS
LIN {X -9.9835,Y -73.2292,Z 80,A -103.4151,B 24.9125,C -2.1605,E1 24.9772,E2 -172.062} C_DIS
LIN {X -12.4125,Y -72.8574,Z 80,A -105.6156,B 24.913,C -2.1534,E1 24.9711,E2 -169.8426} C_DIS
LIN {X -16.2302,Y -72.1034,Z 80,A -108.6426,B 24.913,C -2.1544,E1 24.9628,E2 -166.8145} C_DIS
LIN {X -21.102,Y -70.8303,Z 80,A -113.0879,B 24.9138,C -2.1433,E1 24.9508,E2 -162.3357} C_DIS
LIN {X -24.59,Y -69.6963,Z 80,A -115.2215,B 24.9122,C -2.1634,E1 24.9453,E2 -160.2458} C_DIS
LIN {X -27.9402,Y -68.422,Z 80,A -117.7489,B 24.9115,C -2.1724,E1 24.9387,E2 -157.7342} C_DIS
LIN {X -31.5638,Y -66.8283,Z 80,A -121.6402,B 24.9129,C -2.1554,E1 24.9287,E2 -153.7929} C_DIS
LIN {X -35.9019,Y -64.6011,Z 80,A -124.7513,B 24.9111,C -2.1767,E1 24.9212,E2 -150.7239} C_DIS
LIN {X -38.3119,Y -63.2015,Z 80,A -126.9465,B 24.9109,C -2.179,E1 24.9159,E2 -148.5274} C_DIS
LIN {X -41.0409,Y -61.4652,Z 80,A -129.5533,B 24.9109,C -2.1804,E1 24.9098,E2 -145.9156} C_DIS
LIN {X -43.9772,Y -59.4,Z 80,A -133.2227,B 24.9122,C -2.1638,E1 24.9014,E2 -142.1936} C_DIS
LIN {X -47.1639,Y -56.9016,Z 80,A -135.4526,B 24.9099,C -2.1913,E1 24.8967,E2 -140.0208} C_DIS
LIN {X -49.3949,Y -54.9762,Z 80,A -138.5264,B 24.9111,C -2.1769,E1 24.8902,E2 -136.9007} C_DIS
LIN {X -52.082,Y -52.4378,Z 80,A -140.6737,B 24.9092,C -2.1999,E1 24.886,E2 -134.799} C_DIS
LIN {X -53.9137,Y -50.5524,Z 80,A -143.5696,B 24.9105,C -2.1841,E1 24.8804,E2 -131.8527} C_DIS
LIN {X -56.596,Y -47.5317,Z 80,A -145.5779,B 24.9078,C -2.2175,E1 24.8769,E2 -129.9151} C_DIS
LIN {X -58.1096,Y -45.6676,Z 80,A -147.6916,B 24.9078,C -2.216,E1 24.8732,E2 -127.7877} C_DIS
LIN {X -59.3828,Y -44.0006,Z 80,A -149.9231,B 24.9087,C -2.2057,E1 24.8694,E2 -125.5211} C_DIS
LIN {X -62.0663,Y -40.1255,Z 80,A -152.9598,B 24.9068,C -2.2293,E1 24.8647,E2 -122.5255} C_DIS
LIN {X -63.7785,Y -37.3445,Z 80,A -155.8874,B 24.907,C -2.2267,E1 24.8605,E2 -119.5766} C_DIS
LIN {X -66.3179,Y -32.6204,Z 80,A -159.4524,B 24.9049,C -2.2517,E1 24.856,E2 -116.0524} C_DIS
LIN {X -67.9256,Y -29.1251,Z 80,A -163.2981,B 24.9058,C -2.2403,E1 24.8515,E2 -112.1582} C_DIS
LIN {X -69.6798,Y -24.6368,Z 80,A -166.4337,B 24.9038,C -2.2648,E1 24.8485,E2 -109.0635} C_DIS
LIN {X -70.9598,Y -20.6656,Z 80,A -169.8567,B 24.9033,C -2.2701,E1 24.8457,E2 -105.6334} C_DIS
LIN {X -71.8725,Y -17.219,Z 80,A -172.1699,B 24.9017,C -2.2888,E1 24.8441,E2 -103.3513} C_DIS
LIN {X -72.5141,Y -14.2823,Z 80,A -175.4648,B 24.903,C -2.274,E1 24.8422,E2 -100.0017} C_DIS
LIN {X -73.2747,Y -9.6471,Z 80,A -178.6269,B 24.9011,C -2.2962,E1 24.8409,E2 -96.8736} C_DIS
LIN {X -73.8469,Y -2.9745,Z 80,A 176.553,B 24.8989,C -2.321,E1 24.8399,E2 -92.0838} C_DIS
LIN {X -73.8647,Y 2.4986,Z 80,A 172.2044,B 24.898,C -2.332,E1 24.8399,E2 -87.7354} C_DIS
LIN {X -73.5999,Y 6.7289,Z 80,A 168.7173,B 24.8974,C -2.3379,E1 24.8406,E2 -84.2414} C_DIS
LIN {X -73.2642,Y 9.7277,Z 80,A 166.266,B 24.897,C -2.3428,E1 24.8414,E2 -81.7872} C_DIS
LIN {X -72.7944,Y 12.778,Z 80,A 163.9022,B 24.8963,C -2.351,E1 24.8425,E2 -79.4289} C_DIS
LIN {X -71.9615,Y 16.8467,Z 80,A 160.4904,B 24.8958,C -2.3568,E1 24.8445,E2 -76.0109} C_DIS
LIN {X -70.9862,Y 20.5751,Z 80,A 157.882,B 24.8942,C -2.3747,E1 24.8464,E2 -73.43} C_DIS
LIN {X -70.22,Y 23.0497,Z 80,A 155.7798,B 24.8938,C -2.3788,E1 24.8482,E2 -71.3255} C_DIS
LIN {X -69.4781,Y 25.1993,Z 80,A 153.6766,B 24.894,C -2.3764,E1 24.8501,E2 -69.2048} C_DIS
LIN {X -67.8878,Y 29.2127,Z 80,A 150.0062,B 24.8938,C -2.3792,E1 24.8541,E2 -65.5207} C_DIS
LIN {X -65.3889,Y 34.4454,Z 80,A 145.9417,B 24.8917,C -2.4022,E1 24.8591,E2 -61.4891} C_DIS
LIN {X -63.3071,Y 38.1381,Z 80,A 142.8246,B 24.8905,C -2.4154,E1 24.8634,E2 -58.3874} C_DIS
LIN {X -60.3911,Y 42.6052,Z 80,A 138.7716,B 24.8893,C -2.4287,E1 24.8696,E2 -54.3458} C_DIS
LIN {X -59.138,Y 44.3274,Z 80,A 136.5379,B 24.8901,C -2.4197,E1 24.8734,E2 -52.0799} C_DIS
LIN {X -56.6543,Y 47.4615,Z 80,A 133.8219,B 24.8886,C -2.4366,E1 24.8781,E2 -49.3915} C_DIS
LIN {X -54.6739,Y 49.7288,Z 80,A 131.0555,B 24.889,C -2.4324,E1 24.8833,E2 -46.6028} C_DIS
LIN {X -51.0941,Y 53.4009,Z 80,A 127.2985,B 24.8876,C -2.447,E1 24.8907,E2 -42.8646} C_DIS
LIN {X -49.2082,Y 55.1433,Z 80,A 124.7255,B 24.8885,C -2.4379,E1 24.8961,E2 -40.2598} C_DIS
LIN {X -46.7706,Y 57.2254,Z 80,A 122.6587,B 24.8871,C -2.4531,E1 24.9005,E2 -38.2212} C_DIS
LIN {X -44.0281,Y 59.3613,Z 80,A 120.0313,B 24.8864,C -2.4602,E1 24.9063,E2 -35.6015} C_DIS
LIN {X -41.3187,Y 61.2781,Z 80,A 117.8045,B 24.8852,C -2.4735,E1 24.9114,E2 -33.3987} C_DIS
LIN {X -37.5076,Y 63.6821,Z 80,A 114.3459,B 24.8845,C -2.4808,E1 24.9196,E2 -29.9466} C_DIS
LIN {X -35.784,Y 64.6668,Z 80,A 112.438,B 24.8851,C -2.4746,E1 24.9242,E2 -28.0183} C_DIS
LIN {X -31.3657,Y 66.9212,Z 80,A 108.7541,B 24.8841,C -2.4846,E1 24.9334,E2 -24.3485} C_DIS
LIN {X -28.2407,Y 68.298,Z 80,A 105.9994,B 24.8841,C -2.4858,E1 24.9405,E2 -21.5902} C_DIS
LIN {X -25.3656,Y 69.4176,Z 80,A 103.5652,B 24.8838,C -2.4879,E1 24.9468,E2 -19.1559} C_DIS
LIN {X -22.2751,Y 70.4712,Z 80,A 100.5838,B 24.8846,C -2.4798,E1 24.9548,E2 -16.1499} C_DIS
LIN {X -18.0375,Y 71.6715,Z 80,A 96.9886,B 24.8846,C -2.4788,E1 24.9646,E2 -12.547} C_DIS
LIN {X -14.8526,Y 72.3987,Z 80,A 95.0572,B 24.8831,C -2.4958,E1 24.9697,E2 -10.6537} C_DIS
LIN {X -8.6997,Y 73.3928,Z 80,A 90.2556,B 24.8827,C -2.4998,E1 24.983,E2 -5.8574} C_DIS
LIN {X -5.8677,Y 73.6735,Z 80,A 88.0801,B 24.8825,C -2.5016,E1 24.989,E2 -3.6852} C_DIS
LIN {X -1.5662,Y 73.8905,Z 80,A 84.681,B 24.8825,C -2.5011,E1 24.9985,E2 -0.2843} C_DIS
LIN {X 1.6141,Y 73.8896,Z 80,A 82.4231,B 24.882,C -2.5069,E1 25.0048,E2 1.9598} C_DIS
LIN {X 7.5013,Y 73.525,Z 80,A 77.6951,B 24.8824,C -2.5027,E1 25.018,E2 6.6954} C_DIS
LIN {X 12.7408,Y 72.801,Z 80,A 73.8918,B 24.8818,C -2.5094,E1 25.0284,E2 10.4795} C_DIS
LIN {X 17.626,Y 71.7743,Z 80,A 68.7828,B 24.885,C -2.475,E1 25.0425,E2 15.6632} C_DIS
LIN {X 21.4722,Y 70.7184,Z 80,A 66.6398,B 24.8829,C -2.4978,E1 25.0481,E2 17.7485} C_DIS
LIN {X 25.121,Y 69.5062,Z 80,A 63.6613,B 24.8831,C -2.4953,E1 25.056,E2 20.7269} C_DIS
LIN {X 28.1489,Y 68.3362,Z 80,A 61.1851,B 24.8833,C -2.4939,E1 25.0624,E2 23.201} C_DIS
LIN {X 31.2783,Y 66.9613,Z 80,A 58.664,B 24.8833,C -2.4944,E1 25.0688,E2 25.7146} C_DIS
LIN {X 33.6174,Y 65.8186,Z 80,A 55.8331,B 24.8855,C -2.4699,E1 25.076,E2 28.5958} C_DIS
LIN {X 36.5087,Y 64.2609,Z 80,A 53.8991,B 24.8843,C -2.483,E1 25.0806,E2 30.4931} C_DIS
LIN {X 39.0502,Y 62.748,Z 80,A 51.6667,B 24.8844,C -2.4812,E1 25.0859,E2 32.7228} C_DIS
LIN {X 41.1156,Y 61.4156,Z 80,A 49.2575,B 24.886,C -2.4644,E1 25.0916,E2 35.1638} C_DIS
LIN {X 45.9736,Y 57.8678,Z 80,A 44.5092,B 24.887,C -2.4539,E1 25.1022,E2 39.9197} C_DIS
LIN {X 49.5843,Y 54.8058,Z 80,A 41.4402,B 24.8861,C -2.4634,E1 25.1086,E2 42.954} C_DIS
LIN {X 51.6336,Y 52.8801,Z 80,A 39.2436,B 24.8866,C -2.4585,E1 25.113,E2 45.1533} C_DIS
LIN {X 54.6163,Y 49.793,Z 80,A 35.4651,B 24.8884,C -2.4386,E1 25.1203,E2 48.9622} C_DIS
LIN {X 57.0856,Y 46.9414,Z 80,A 32.2421,B 24.8898,C -2.4235,E1 25.126,E2 52.2062} C_DIS
LIN {X 59.3976,Y 43.9806,Z 80,A 30.1184,B 24.8884,C -2.4387,E1 25.1295,E2 54.2838} C_DIS
LIN {X 61.2333,Y 41.3848,Z 80,A 27.6682,B 24.8889,C -2.4329,E1 25.1334,E2 56.7356} C_DIS
LIN {X 62.9607,Y 38.708,Z 80,A 25.5191,B 24.8887,C -2.4357,E1 25.1366,E2 58.8672} C_DIS
LIN {X 65.0299,Y 35.1191,Z 80,A 22.1586,B 24.8898,C -2.4229,E1 25.1413,E2 62.2407} C_DIS
LIN {X 66.4563,Y 32.339,Z 80,A 19.6114,B 24.8908,C -2.4126,E1 25.1445,E2 64.7985} C_DIS
LIN {X 67.6376,Y 29.7899,Z 80,A 17.3994,B 24.8914,C -2.4055,E1 25.147,E2 67.0152} C_DIS
LIN {X 68.5268,Y 27.6828,Z 80,A 15.4659,B 24.8923,C -2.3958,E1 25.1491,E2 68.961} C_DIS
LIN {X 69.6155,Y 24.8162,Z 80,A 12.3855,B 24.8947,C -2.3687,E1 25.152,E2 72.0882} C_DIS
LIN {X 70.9166,Y 20.8112,Z 80,A 10.0595,B 24.8932,C -2.386,E1 25.1538,E2 74.3602} C_DIS
LIN {X 71.9474,Y 16.9014,Z 80,A 6.8696,B 24.8942,C -2.3749,E1 25.156,E2 77.5579} C_DIS
LIN {X 72.6842,Y 13.3837,Z 80,A 3.8943,B 24.8954,C -2.3608,E1 25.1576,E2 80.5491} C_DIS
LIN {X 73.1891,Y 10.276,Z 80,A 1.7872,B 24.8952,C -2.3629,E1 25.1585,E2 82.6387} C_DIS
LIN {X 73.578,Y 6.9627,Z 80,A -0.7914,B 24.8959,C -2.355,E1 25.1592,E2 85.2207} C_DIS
LIN {X 73.8044,Y 3.8877,Z 80,A -3.1536,B 24.8965,C -2.3483,E1 25.1596,E2 87.5848} C_DIS
LIN {X 73.8912,Y 1.5285,Z 80,A -4.9262,B 24.8969,C -2.3442,E1 25.1598,E2 89.3567} C_DIS
LIN {X 73.8873,Y -1.7088,Z 80,A -7.5014,B 24.8978,C -2.3343,E1 25.1597,E2 91.9398} C_DIS
LIN {X 73.7405,Y -4.9553,Z 80,A -9.9939,B 24.8984,C -2.327,E1 25.1593,E2 94.4347} C_DIS
LIN {X 73.4477,Y -8.2258,Z 80,A -12.3613,B 24.8987,C -2.3241,E1 25.1587,E2 96.7949} C_DIS
LIN {X 72.9334,Y -11.9577,Z 80,A -15.3723,B 24.8997,C -2.3122,E1 25.1574,E2 99.8163} C_DIS
LIN {X 72.102,Y -16.2365,Z 80,A -18.8216,B 24.9008,C -2.2995,E1 25.1555,E2 103.2756} C_DIS
LIN {X 71.3172,Y -19.3932,Z 80,A -21.3039,B 24.9014,C -2.2927,E1 25.1537,E2 105.7596} C_DIS
LIN {X 70.2565,Y -22.9404,Z 80,A -24.916,B 24.904,C -2.2623,E1 25.1506,E2 109.423} C_DIS
LIN {X 68.9733,Y -26.5527,Z 80,A -26.8994,B 24.9023,C -2.2819,E1 25.1487,E2 111.349} C_DIS
LIN {X 67.6222,Y -29.8248,Z 80,A -29.4773,B 24.9026,C -2.2785,E1 25.146,E2 113.9208} C_DIS
LIN {X 65.6172,Y -34.0082,Z 80,A -33.2739,B 24.904,C -2.262,E1 25.1413,E2 117.736} C_DIS
LIN {X 63.376,Y -38.0242,Z 80,A -36.9451,B 24.9051,C -2.2487,E1 25.1362,E2 121.4196} C_DIS
LIN {X 61.5779,Y -40.8709,Z 80,A -40.4538,B 24.9079,C -2.2156,E1 25.1307,E2 124.989} C_DIS
LIN {X 59.1552,Y -44.3046,Z 80,A -44.0098,B 24.9093,C -2.1984,E1 25.1247,E2 128.5687} C_DIS
LIN {X 55.9639,Y -48.2734,Z 80,A -46.3538,B 24.9064,C -2.234,E1 25.1207,E2 130.8179} C_DIS
LIN {X 53.6535,Y -50.8275,Z 80,A -49.528,B 24.9081,C -2.2128,E1 25.1146,E2 134.028} C_DIS
LIN {X 50.5879,Y -53.8798,Z 80,A -53.1673,B 24.9095,C -2.1968,E1 25.1072,E2 137.6902} C_DIS
LIN {X 47.7523,Y -56.4092,Z 80,A -55.9114,B 24.9095,C -2.1959,E1 25.1014,E2 140.4258} C_DIS
LIN {X 43.9529,Y -59.4179,Z 80,A -59.0157,B 24.9087,C -2.2063,E1 25.0947,E2 143.4939} C_DIS
LIN {X 41.395,Y -61.2264,Z 80,A -61.7393,B 24.9098,C -2.1931,E1 25.0884,E2 146.2393} C_DIS
LIN {X 39.4522,Y -62.4969,Z 80,A -63.6583,B 24.9103,C -2.1864,E1 25.0838,E2 148.1682} C_DIS
LIN {X 36.365,Y -64.3424,Z 80,A -66.3906,B 24.9106,C -2.1829,E1 25.0772,E2 150.9004} C_DIS
LIN {X 33.438,Y -65.9103,Z 80,A -68.9383,B 24.9109,C -2.1794,E1 25.0709,E2 153.4494} C_DIS
LIN {X 30.2491,Y -67.4331,Z 80,A -71.2438,B 24.9103,C -2.1872,E1 25.0652,E2 155.7305} C_DIS
LIN {X 27.2669,Y -68.6935,Z 80,A -73.7217,B 24.9105,C -2.1844,E1 25.0588,E2 158.2091} C_DIS
LIN {X 24.0339,Y -69.8912,Z 80,A -76.9566,B 24.912,C -2.1655,E1 25.0502,E2 161.4822} C_DIS
LIN {X 20.4357,Y -71.0259,Z 80,A -79.7548,B 24.912,C -2.1656,E1 25.0427,E2 164.2751} C_DIS
LIN {X 17.2139,Y -71.8737,Z 80,A -82.2831,B 24.9121,C -2.1645,E1 25.0359,E2 166.8022} C_DIS
LIN {X 14.8664,Y -72.3959,Z 80,A -84.9432,B 24.914,C -2.1416,E1 25.0285,E2 169.5135} C_DIS
LIN {X 11.1013,Y -73.0686,Z 80,A -86.7095,B 24.9116,C -2.1715,E1 25.0238,E2 171.2071} C_DIS
LIN {X 8.1934,Y -73.4512,Z 80,A -89.3607,B 24.9125,C -2.1599,E1 25.0164,E2 173.8837} C_DIS
LIN {X 5.0638,Y -73.7332,Z 80,A -91.8162,B 24.9126,C -2.1582,E1 25.0095,E2 176.3419} C_DIS
LIN {X 1.7403,Y -73.8864,Z 80,A -94.97,B 24.9139,C -2.1422,E1 25.0006,E2 179.5329} C_DIS
LIN {X 1.7403,Y -73.8864,Z 80,A -94.97,B 24.9139,C -2.1422,E1 25.0006,E2 179.5329} C_DIS
Enddeposition()
LIN {X 0.4724,Y -73.0059,Z 80,A -94.7223,B 24.91,C -2.1901,E1 25.0016,E2 179.1716} C_DIS
Startdeposition()
$VEL.CP = VEL_PRINT
LIN {X 3.1492,Y -72.9448,Z 80,A -92.1368,B 24.9089,C -2.2035,E1 25.0089,E2 176.5548} C_DIS
LIN {X 6.0764,Y -72.7597,Z 80,A -89.8459,B 24.9089,C -2.2043,E1 25.0153,E2 174.2632} C_DIS
LIN {X 9.1865,Y -72.4328,Z 80,A -87.3594,B 24.9087,C -2.2067,E1 25.0222,E2 171.7729} C_DIS
LIN {X 14.0285,Y -71.6528,Z 80,A -83.5844,B 24.9086,C -2.2076,E1 25.0326,E2 167.9997} C_DIS
LIN {X 16.8822,Y -71.0339,Z 80,A -81.2266,B 24.9083,C -2.2115,E1 25.039,E2 165.6358} C_DIS
LIN {X 20.3405,Y -70.1234,Z 80,A -78.4219,B 24.908,C -2.2145,E1 25.0466,E2 162.8287} C_DIS
LIN {X 23.2857,Y -69.2,Z 80,A -76.103,B 24.908,C -2.2145,E1 25.0527,E2 160.514} C_DIS
LIN {X 26.9321,Y -67.8644,Z 80,A -73.2697,B 24.9082,C -2.2127,E1 25.0601,E2 157.6911} C_DIS
LIN {X 29.0584,Y -66.9808,Z 80,A -71.5622,B 24.9082,C -2.2125,E1 25.0645,E2 155.988} C_DIS
LIN {X 31.0894,Y -66.0636,Z 80,A -69.3727,B 24.9069,C -2.2275,E1 25.0701,E2 153.7686} C_DIS
LIN {X 34.2073,Y -64.504,Z 80,A -66.7563,B 24.9069,C -2.2287,E1 25.0766,E2 151.1566} C_DIS
LIN {X 38.87,Y -61.8064,Z 80,A -62.4722,B 24.906,C -2.238,E1 25.0869,E2 146.8637} C_DIS
LIN {X 41.6739,Y -59.9512,Z 80,A -59.8483,B 24.9056,C -2.2428,E1 25.093,E2 144.2374} C_DIS
LIN {X 44.5958,Y -57.8107,Z 80,A -56.3951,B 24.9036,C -2.2663,E1 25.1007,E2 140.7411} C_DIS
LIN {X 47.2298,Y -55.6798,Z 80,A -54.4052,B 24.9048,C -2.2529,E1 25.1049,E2 138.7906} C_DIS
LIN {X 51.409,Y -51.8459,Z 80,A -50.5781,B 24.9054,C -2.2454,E1 25.1127,E2 134.9967} C_DIS
LIN {X 53.2697,Y -49.9321,Z 80,A -47.5941,B 24.9028,C -2.2761,E1 25.1186,E2 131.953} C_DIS
LIN {X 55.8592,Y -47.019,Z 80,A -44.3256,B 24.9016,C -2.29,E1 25.1245,E2 128.6664} C_DIS
LIN {X 59.0658,Y -42.9205,Z 80,A -40.5983,B 24.9016,C -2.2905,E1 25.1308,E2 124.9557} C_DIS
LIN {X 60.9422,Y -40.2108,Z 80,A -38.2586,B 24.9016,C -2.2905,E1 25.1344,E2 122.6278} C_DIS
LIN {X 62.6542,Y -37.4887,Z 80,A -35.6909,B 24.9008,C -2.2989,E1 25.1382,E2 120.0532} C_DIS
LIN {X 64.4875,Y -34.2387,Z 80,A -31.5777,B 24.897,C -2.3425,E1 25.1437,E2 115.8587} C_DIS
LIN {X 66.6526,Y -29.805,Z 80,A -29.3962,B 24.9004,C -2.304,E1 25.1461,E2 113.7799} C_DIS
LIN {X 67.5056,Y -27.8177,Z 80,A -27.3327,B 24.899,C -2.3199,E1 25.1484,E2 111.6902} C_DIS
LIN {X 68.816,Y -24.397,Z 80,A -24.8697,B 24.8993,C -2.3166,E1 25.1508,E2 109.2487} C_DIS
LIN {X 69.5886,Y -22.1008,Z 80,A -22.4927,B 24.8976,C -2.3364,E1 25.1529,E2 106.8383} C_DIS
LIN {X 70.4776,Y -19.0729,Z 80,A -20.0697,B 24.897,C -2.3426,E1 25.1547,E2 104.4146} C_DIS
LIN {X 71.2163,Y -16.1005,Z 80,A -17.6985,B 24.8965,C -2.3492,E1 25.1562,E2 102.0416} C_DIS
LIN {X 71.9499,Y -12.4186,Z 80,A -15.0547,B 24.8965,C -2.3496,E1 25.1576,E2 99.4123} C_DIS
LIN {X 72.2617,Y -10.446,Z 80,A -13.0671,B 24.8949,C -2.367,E1 25.1584,E2 97.3954} C_DIS
LIN {X 72.667,Y -7.0926,Z 80,A -10.5937,B 24.8946,C -2.3702,E1 25.1592,E2 94.929} C_DIS
LIN {X 72.9072,Y -3.9208,Z 80,A -8.1209,B 24.8939,C -2.3774,E1 25.1596,E2 92.4537} C_DIS
LIN {X 73.0094,Y -0.7704,Z 80,A -5.6798,B 24.8933,C -2.3843,E1 25.1598,E2 90.0109} C_DIS
LIN {X 72.9955,Y 1.6059,Z 80,A -3.806,B 24.8928,C -2.3905,E1 25.1597,E2 88.1335} C_DIS
LIN {X 72.8801,Y 4.4049,Z 80,A -1.5594,B 24.892,C -2.3989,E1 25.1594,E2 85.8805} C_DIS
LIN {X 72.618,Y 7.582,Z 80,A 0.9986,B 24.8911,C -2.4084,E1 25.1587,E2 83.3152} C_DIS
LIN {X 72.2805,Y 10.315,Z 80,A 3.3585,B 24.89,C -2.421,E1 25.1578,E2 80.9394} C_DIS
LIN {X 71.5018,Y 14.7775,Z 80,A 6.3506,B 24.8905,C -2.4154,E1 25.1563,E2 77.978} C_DIS
LIN {X 71.0144,Y 16.963,Z 80,A 8.3218,B 24.8894,C -2.4271,E1 25.155,E2 75.9908} C_DIS
LIN {X 70.0368,Y 20.6332,Z 80,A 12.2076,B 24.8862,C -2.4627,E1 25.1519,E2 72.0432} C_DIS
LIN {X 68.759,Y 24.5559,Z 80,A 14.3718,B 24.8882,C -2.4406,E1 25.15,E2 69.9431} C_DIS
LIN {X 67.6754,Y 27.4031,Z 80,A 16.8594,B 24.8873,C -2.4503,E1 25.1475,E2 67.4465} C_DIS
LIN {X 66.4735,Y 30.2024,Z 80,A 19.2235,B 24.8868,C -2.4563,E1 25.1448,E2 65.0812} C_DIS
LIN {X 65.1179,Y 33.024,Z 80,A 21.7287,B 24.886,C -2.4645,E1 25.1417,E2 62.5699} C_DIS
LIN {X 63.3811,Y 36.2453,Z 80,A 24.3264,B 24.886,C -2.4643,E1 25.1382,E2 59.9863} C_DIS
LIN {X 62.06,Y 38.4641,Z 80,A 26.4652,B 24.8852,C -2.4728,E1 25.1351,E2 57.8383} C_DIS
LIN {X 60.5989,Y 40.7272,Z 80,A 28.5714,B 24.8848,C -2.4779,E1 25.1319,E2 55.7304} C_DIS
LIN {X 58.8755,Y 43.1804,Z 80,A 30.9793,B 24.8841,C -2.4853,E1 25.1279,E2 53.3168} C_DIS
LIN {X 56.3206,Y 46.4642,Z 80,A 34.2287,B 24.8834,C -2.4926,E1 25.1223,E2 50.0654} C_DIS
LIN {X 54.2186,Y 48.9006,Z 80,A 37.5903,B 24.8806,C -2.5221,E1 25.1159,E2 46.6489} C_DIS
LIN {X 51.5477,Y 51.7086,Z 80,A 39.458,B 24.8831,C -2.4952,E1 25.1124,E2 44.8527} C_DIS
LIN {X 50.2787,Y 52.9437,Z 80,A 41.1566,B 24.882,C -2.5067,E1 25.1089,E2 43.134} C_DIS
LIN {X 47.8662,Y 55.1338,Z 80,A 43.8889,B 24.8811,C -2.5167,E1 25.1032,E2 40.389} C_DIS
LIN {X 44.9703,Y 57.5211,Z 80,A 46.6847,B 24.881,C -2.5179,E1 25.0971,E2 37.6008} C_DIS
LIN {X 40.9562,Y 60.4438,Z 80,A 50.4284,B 24.8808,C -2.5202,E1 25.0886,E2 33.8647} C_DIS
LIN {X 38.4065,Y 62.096,Z 80,A 52.9648,B 24.88,C -2.528,E1 25.0826,E2 31.3179} C_DIS
LIN {X 35.755,Y 63.659,Z 80,A 55.2315,B 24.88,C -2.5273,E1 25.0771,E2 29.0596} C_DIS
LIN {X 32.6978,Y 65.2825,Z 80,A 57.9211,B 24.8798,C -2.5301,E1 25.0705,E2 26.371} C_DIS
LIN {X 29.2852,Y 66.8824,Z 80,A 60.7914,B 24.8798,C -2.5311,E1 25.0632,E2 23.5055} C_DIS
LIN {X 26.7499,Y 67.9361,Z 80,A 63.0737,B 24.8792,C -2.5367,E1 25.0573,E2 21.2151} C_DIS
LIN {X 23.8816,Y 68.9973,Z 80,A 65.5826,B 24.8787,C -2.5418,E1 25.0506,E2 18.6994} C_DIS
LIN {X 20.8832,Y 69.9627,Z 80,A 68.2057,B 24.8782,C -2.5477,E1 25.0436,E2 16.0669} C_DIS
LIN {X 17.8053,Y 70.808,Z 80,A 70.439,B 24.8787,C -2.542,E1 25.0376,E2 13.8507} C_DIS
LIN {X 14.7537,Y 71.5066,Z 80,A 72.923,B 24.8785,C -2.5439,E1 25.0308,E2 11.3654} C_DIS
LIN {X 11.7369,Y 72.0638,Z 80,A 76.078,B 24.8765,C -2.5644,E1 25.022,E2 8.1647} C_DIS
LIN {X 8.1994,Y 72.5512,Z 80,A 77.85,B 24.8791,C -2.5379,E1 25.0173,E2 6.4571} C_DIS
LIN {X 2.3402,Y 72.9753,Z 80,A 82.7023,B 24.8785,C -2.5442,E1 25.0038,E2 1.592} C_DIS
LIN {X -0.5939,Y 73.0105,Z 80,A 85.0998,B 24.8783,C -2.5462,E1 24.997,E2 -0.8102} C_DIS
LIN {X -4.1574,Y 72.8944,Z 80,A 87.9017,B 24.8783,C -2.5453,E1 24.9892,E2 -3.6106} C_DIS
LIN {X -6.9502,Y 72.6809,Z 80,A 89.9635,B 24.8788,C -2.5408,E1 24.9835,E2 -5.6628} C_DIS
LIN {X -11.7477,Y 72.062,Z 80,A 93.5613,B 24.8795,C -2.5334,E1 24.9736,E2 -9.2458} C_DIS
LIN {X -14.095,Y 71.64,Z 80,A 95.7517,B 24.8789,C -2.54,E1 24.9675,E2 -11.4541} C_DIS
LIN {X -17.7901,Y 70.8118,Z 80,A 99.2393,B 24.8779,C -2.5501,E1 24.958,E2 -14.9706} C_DIS
LIN {X -22.0277,Y 69.6118,Z 80,A 101.8895,B 24.8802,C -2.5263,E1 24.9511,E2 -17.5685} C_DIS
LIN {X -25.4041,Y 68.4502,Z 80,A 104.9327,B 24.88,C -2.5288,E1 24.943,E2 -20.6236} C_DIS
LIN {X -28.3626,Y 67.2787,Z 80,A 107.5656,B 24.88,C -2.5286,E1 24.9362,E2 -23.2621} C_DIS
LIN {X -31.5268,Y 65.8554,Z 80,A 110.3325,B 24.8803,C -2.5256,E1 24.9292,E2 -26.0286} C_DIS
LIN {X -34.6817,Y 64.25,Z 80,A 113.4043,B 24.88,C -2.5281,E1 24.9216,E2 -29.115} C_DIS
LIN {X -38.2417,Y 62.1979,Z 80,A 116.4437,B 24.881,C -2.5178,E1 24.9143,E2 -32.1391} C_DIS
LIN {X -41.1966,Y 60.2806,Z 80,A 119.0889,B 24.8818,C -2.5097,E1 24.9082,E2 -34.7736} C_DIS
LIN {X -44.29,Y 58.046,Z 80,A 121.7464,B 24.8831,C -2.4955,E1 24.9023,E2 -37.4068} C_DIS
LIN {X -46.7603,Y 56.0745,Z 80,A 124.8197,B 24.8823,C -2.5042,E1 24.8956,E2 -40.5126} C_DIS
LIN {X -48.9595,Y 54.1654,Z 80,A 126.8238,B 24.8834,C -2.4924,E1 24.8914,E2 -42.4963} C_DIS
LIN {X -51.2607,Y 51.9924,Z 80,A 129.3438,B 24.8839,C -2.4874,E1 24.8864,E2 -45.015} C_DIS
LIN {X -53.2082,Y 49.9974,Z 80,A 131.9089,B 24.8835,C -2.491,E1 24.8814,E2 -47.5997} C_DIS
LIN {X -55.649,Y 47.2659,Z 80,A 134.4127,B 24.885,C -2.475,E1 24.8769,E2 -50.0768} C_DIS
LIN {X -57.6033,Y 44.865,Z 80,A 137.199,B 24.8848,C -2.477,E1 24.872,E2 -52.8808} C_DIS
LIN {X -59.636,Y 42.1248,Z 80,A 140.6214,B 24.8839,C -2.4872,E1 24.8665,E2 -56.3445} C_DIS
LIN {X -62.1013,Y 38.398,Z 80,A 142.9489,B 24.8873,C -2.4499,E1 24.8631,E2 -58.5948} C_DIS
LIN {X -63.4845,Y 36.0654,Z 80,A 145.1535,B 24.8877,C -2.4457,E1 24.86,E2 -60.8006} C_DIS
LIN {X -64.7453,Y 33.7475,Z 80,A 147.818,B 24.887,C -2.4534,E1 24.8565,E2 -63.4976} C_DIS
LIN {X -66.7456,Y 29.5974,Z 80,A 151.0461,B 24.8888,C -2.4337,E1 24.8528,E2 -66.6964} C_DIS
LIN {X -67.9734,Y 26.6548,Z 80,A 153.5049,B 24.8896,C -2.4251,E1 24.8502,E2 -69.1486} C_DIS
LIN {X -69.619,Y 22.0023,Z 80,A 157.1723,B 24.8911,C -2.4086,E1 24.8469,E2 -72.7972} C_DIS
LIN {X -70.2137,Y 20.023,Z 80,A 159.0063,B 24.8911,C -2.4084,E1 24.8455,E2 -74.6413} C_DIS
LIN {X -71.0645,Y 16.7546,Z 80,A 161.6318,B 24.892,C -2.3995,E1 24.8437,E2 -77.2611} C_DIS
LIN {X -71.7343,Y 13.6052,Z 80,A 164.2381,B 24.8925,C -2.3934,E1 24.8423,E2 -79.868} C_DIS
LIN {X -72.2545,Y 10.4976,Z 80,A 166.6668,B 24.8933,C -2.3845,E1 24.8412,E2 -82.2901} C_DIS
LIN {X -72.6266,Y 7.5001,Z 80,A 169.0881,B 24.8939,C -2.3782,E1 24.8405,E2 -84.7107} C_DIS
LIN {X -72.9377,Y 3.3153,Z 80,A 172.0066,B 24.8956,C -2.3592,E1 24.8399,E2 -87.6013} C_DIS
LIN {X -73.0105,Y -0.5663,Z 80,A 174.9593,B 24.8966,C -2.3474,E1 24.8399,E2 -90.5436} C_DIS
LIN {X -72.9605,Y -2.7511,Z 80,A 177.1271,B 24.8962,C -2.3522,E1 24.8399,E2 -92.736} C_DIS
LIN {X -72.7023,Y -6.7266,Z 80,A -179.6884,B 24.8969,C -2.3437,E1 24.8406,E2 -95.9192} C_DIS
LIN {X -72.3464,Y -9.8477,Z 80,A -177.1742,B 24.8975,C -2.3371,E1 24.8415,E2 -98.4327} C_DIS
LIN {X -71.8881,Y -12.767,Z 80,A -174.7096,B 24.8979,C -2.3332,E1 24.8427,E2 -100.9028} C_DIS
LIN {X -71.293,Y -15.7549,Z 80,A -172.4782,B 24.8988,C -2.3223,E1 24.8439,E2 -103.1212} C_DIS
LIN {X -70.657,Y -18.3987,Z 80,A -170.2417,B 24.8992,C -2.3182,E1 24.8455,E2 -105.361} C_DIS
LIN {X -69.7365,Y -21.6258,Z 80,A -167.6007,B 24.8998,C -2.3105,E1 24.8476,E2 -107.9989} C_DIS
LIN {X -68.7858,Y -24.4811,Z 80,A -165.2653,B 24.9005,C -2.303,E1 24.8497,E2 -110.3296} C_DIS
LIN {X -67.0672,Y -28.8578,Z 80,A -161.9674,B 24.9022,C -2.2833,E1 24.8531,E2 -113.599} C_DIS
LIN {X -66.1437,Y -30.9175,Z 80,A -159.807,B 24.9018,C -2.2874,E1 24.8556,E2 -115.7809} C_DIS
LIN {X -64.8776,Y -33.494,Z 80,A -157.501,B 24.9023,C -2.2824,E1 24.8585,E2 -118.0875} C_DIS
LIN {X -62.6914,Y -37.4262,Z 80,A -153.9358,B 24.903,C -2.2739,E1 24.8635,E2 -121.6509} C_DIS
LIN {X -61.0873,Y -39.9908,Z 80,A -151.5403,B 24.9035,C -2.2683,E1 24.8671,E2 -124.0453} C_DIS
LIN {X -59.2775,Y -42.6276,Z 80,A -149.1895,B 24.9043,C -2.2584,E1 24.8708,E2 -126.3838} C_DIS
LIN {X -57.6961,Y -44.7445,Z 80,A -146.8951,B 24.9043,C -2.2586,E1 24.8747,E2 -128.6898} C_DIS
LIN {X -55.6803,Y -47.2292,Z 80,A -144.5042,B 24.905,C -2.25,E1 24.879,E2 -131.0712} C_DIS
LIN {X -53.225,Y -49.9797,Z 80,A -141.6419,B 24.9056,C -2.2429,E1 24.8843,E2 -133.9292} C_DIS
LIN {X -51.2258,Y -52.0269,Z 80,A -139.1061,B 24.9054,C -2.2452,E1 24.8894,E2 -136.4812} C_DIS
LIN {X -49.0381,Y -54.0943,Z 80,A -136.8368,B 24.906,C -2.2382,E1 24.894,E2 -138.7432} C_DIS
LIN {X -46.6312,Y -56.1818,Z 80,A -134.3608,B 24.9065,C -2.233,E1 24.8993,E2 -141.2162} C_DIS
LIN {X -43.4877,Y -58.6501,Z 80,A -131.1341,B 24.9067,C -2.2296,E1 24.9064,E2 -144.4466} C_DIS
LIN {X -40.883,Y -60.4934,Z 80,A -128.77,B 24.9074,C -2.2222,E1 24.9118,E2 -146.801} C_DIS
LIN {X -38.4892,Y -62.0443,Z 80,A -126.5179,B 24.9076,C -2.2191,E1 24.9171,E2 -149.0529} C_DIS
LIN {X -35.9296,Y -63.5615,Z 80,A -124.228,B 24.908,C -2.2147,E1 24.9227,E2 -151.3392} C_DIS
LIN {X -32.8827,Y -65.1886,Z 80,A -121.3805,B 24.908,C -2.2147,E1 24.9297,E2 -154.1945} C_DIS
LIN {X -29.9748,Y -66.5758,Z 80,A -118.7467,B 24.908,C -2.2145,E1 24.9364,E2 -156.8344} C_DIS
LIN {X -26.8249,Y -67.9066,Z 80,A -116.1897,B 24.9085,C -2.2087,E1 24.943,E2 -159.3832} C_DIS
LIN {X -23.789,Y -69.0298,Z 80,A -113.3184,B 24.908,C -2.2149,E1 24.9506,E2 -162.275} C_DIS
LIN {X -20.5972,Y -70.0475,Z 80,A -111.0142,B 24.9088,C -2.2048,E1 24.9567,E2 -164.559} C_DIS
LIN {X -17.7204,Y -70.8294,Z 80,A -108.5672,B 24.9088,C -2.2062,E1 24.9634,E2 -167.013} C_DIS
LIN {X -11.5123,Y -72.1004,Z 80,A -103.9698,B 24.9097,C -2.1945,E1 24.9759,E2 -171.5876} C_DIS
LIN {X -8.2091,Y -72.5499,Z 80,A -100.6233,B 24.9081,C -2.2132,E1 24.9853,E2 -174.981} C_DIS
LIN {X -4.7551,Y -72.8575,Z 80,A -98.3753,B 24.9092,C -2.2007,E1 24.9915,E2 -177.2001} C_DIS
LIN {X -1.7773,Y -72.9911,Z 80,A -96.041,B 24.9092,C -2.2008,E1 24.998,E2 -179.5351} C_DIS
LIN {X 0.4724,Y -73.0059,Z 80,A -94.721,B 24.9101,C -2.1895,E1 25.0016,E2 -180.8284} C_DIS
Enddeposition()
LIN {X 0.4724,Y -73.0059,Z 80,A -94.721,B 24.9101,C -2.1895,E1 25.0016,E2 -180.8284} C_DIS
Startdeposition()
$VEL.CP = VEL_PRINT
LIN {X -0.0115,Y -72.12,Z 80,A -95.7491,B 24.9101,C -2.1882,E1 24.9987,E2 -179.7971} C_DIS
LIN {X -2.6597,Y -72.0693,Z 80,A -97.79,B 24.9101,C -2.1895,E1 24.993,E2 -177.7592} C_DIS
LIN {X -5.4918,Y -71.909,Z 80,A -100.0153,B 24.9101,C -2.1902,E1 24.9868,E2 -175.5346} C_DIS
LIN {X -8.3828,Y -71.6298,Z 80,A -102.3676,B 24.9101,C -2.1893,E1 24.9803,E2 -173.1788} C_DIS
LIN {X -11.1983,Y -71.2442,Z 80,A -104.7493,B 24.9103,C -2.1867,E1 24.9737,E2 -170.7889} C_DIS
LIN {X -14.1105,Y -70.7249,Z 80,A -107.0216,B 24.9101,C -2.1895,E1 24.9675,E2 -168.5209} C_DIS
LIN {X -16.6834,Y -70.1621,Z 80,A -109.2165,B 24.9102,C -2.188,E1 24.9615,E2 -166.3195} C_DIS
LIN {X -20.0879,Y -69.2658,Z 80,A -112.0541,B 24.9102,C -2.1887,E1 24.9538,E2 -163.4791} C_DIS
LIN {X -23.4659,Y -68.1956,Z 80,A -114.9342,B 24.9101,C -2.1893,E1 24.9462,E2 -160.5952} C_DIS
LIN {X -26.3087,Y -67.1488,Z 80,A -117.1716,B 24.9096,C -2.1957,E1 24.9404,E2 -158.3682} C_DIS
LIN {X -28.9704,Y -66.0443,Z 80,A -119.5482,B 24.9096,C -2.1959,E1 24.9343,E2 -155.9867} C_DIS
LIN {X -31.6836,Y -64.786,Z 80,A -121.7596,B 24.909,C -2.2027,E1 24.9287,E2 -153.7858} C_DIS
LIN {X -34.0064,Y -63.5985,Z 80,A -123.9345,B 24.909,C -2.2028,E1 24.9233,E2 -151.6052} C_DIS
LIN {X -36.6484,Y -62.1128,Z 80,A -126.2835,B 24.9086,C -2.2076,E1 24.9176,E2 -149.2606} C_DIS
LIN {X -39.0206,Y -60.6507,Z 80,A -128.6328,B 24.9086,C -2.2076,E1 24.9121,E2 -146.9041} C_DIS
LIN {X -41.5271,Y -58.9633,Z 80,A -130.9192,B 24.908,C -2.2143,E1 24.9068,E2 -144.6256} C_DIS
LIN {X -43.6818,Y -57.3858,Z 80,A -133.1675,B 24.908,C -2.2149,E1 24.9018,E2 -142.3709} C_DIS
LIN {X -46.2393,Y -55.345,Z 80,A -135.7719,B 24.9076,C -2.2196,E1 24.8962,E2 -139.7678} C_DIS
LIN {X -48.6163,Y -53.2691,Z 80,A -138.2434,B 24.9071,C -2.2253,E1 24.891,E2 -137.3} C_DIS
LIN {X -50.8656,Y -51.126,Z 80,A -140.7532,B 24.9068,C -2.2294,E1 24.886,E2 -134.7895} C_DIS
LIN {X -52.9785,Y -48.9331,Z 80,A -143.1846,B 24.9064,C -2.2343,E1 24.8813,E2 -132.3593} C_DIS
LIN {X -55.1895,Y -46.4264,Z 80,A -145.9419,B 24.906,C -2.238,E1 24.8763,E2 -129.5981} C_DIS
LIN {X -57.2388,Y -43.8733,Z 80,A -148.5098,B 24.9055,C -2.2449,E1 24.8719,E2 -127.0347} C_DIS
LIN {X -59.1805,Y -41.2163,Z 80,A -151.0065,B 24.9047,C -2.254,E1 24.8678,E2 -124.5475} C_DIS
LIN {X -60.9305,Y -38.5844,Z 80,A -153.5764,B 24.9043,C -2.259,E1 24.8639,E2 -121.9766} C_DIS
LIN {X -62.3248,Y -36.289,Z 80,A -155.7005,B 24.9038,C -2.2648,E1 24.8609,E2 -119.8554} C_DIS
LIN {X -63.6102,Y -33.9847,Z 80,A -157.8435,B 24.9034,C -2.2694,E1 24.858,E2 -117.712} C_DIS
LIN {X -64.8114,Y -31.6319,Z 80,A -159.9326,B 24.9029,C -2.2754,E1 24.8554,E2 -115.626} C_DIS
LIN {X -65.9273,Y -29.2372,Z 80,A -162.2207,B 24.9027,C -2.277,E1 24.8528,E2 -113.3292} C_DIS
LIN {X -67.139,Y -26.3337,Z 80,A -164.6573,B 24.902,C -2.2856,E1 24.8502,E2 -110.8994} C_DIS
LIN {X -68.2342,Y -23.3516,Z 80,A -167.1852,B 24.9014,C -2.2928,E1 24.8479,E2 -108.3746} C_DIS
LIN {X -69.268,Y -20.08,Z 80,A -169.9878,B 24.9008,C -2.2992,E1 24.8456,E2 -105.5711} C_DIS
LIN {X -70.1665,Y -16.6655,Z 80,A -172.6777,B 24.8999,C -2.3103,E1 24.8438,E2 -102.8919} C_DIS
LIN {X -70.8083,Y -13.6854,Z 80,A -175.0663,B 24.8991,C -2.3185,E1 24.8424,E2 -100.5087} C_DIS
LIN {X -71.2625,Y -11.0795,Z 80,A -177.1927,B 24.8986,C -2.3244,E1 24.8415,E2 -98.3839} C_DIS
LIN {X -71.6371,Y -8.3209,Z 80,A -179.4145,B 24.898,C -2.3311,E1 24.8407,E2 -96.1648} C_DIS
LIN {X -71.885,Y -5.7995,Z 80,A 178.532,B 24.8976,C -2.3365,E1 24.8402,E2 -94.112} C_DIS
LIN {X -72.0493,Y -3.1643,Z 80,A 176.4059,B 24.897,C -2.3425,E1 24.8399,E2 -91.9873} C_DIS
LIN {X -72.118,Y -0.2837,Z 80,A 174.0645,B 24.8965,C -2.3486,E1 24.8398,E2 -89.6465} C_DIS
LIN {X -72.0694,Y 2.6569,Z 80,A 171.7196,B 24.8959,C -2.3559,E1 24.84,E2 -87.3047} C_DIS
LIN {X -71.882,Y 5.8374,Z 80,A 169.2446,B 24.895,C -2.3651,E1 24.8404,E2 -84.837} C_DIS
LIN {X -71.6358,Y 8.3324,Z 80,A 167.2248,B 24.8945,C -2.3709,E1 24.841,E2 -82.8188} C_DIS
LIN {X -71.2609,Y 11.0907,Z 80,A 164.8806,B 24.8942,C -2.375,E1 24.842,E2 -80.4704} C_DIS
LIN {X -70.7345,Y 14.0634,Z 80,A 162.5451,B 24.8934,C -2.3839,E1 24.8432,E2 -78.1424} C_DIS
LIN {X -70.1657,Y 16.6685,Z 80,A 160.3154,B 24.893,C -2.3881,E1 24.8446,E2 -75.9097} C_DIS
LIN {X -69.2661,Y 20.0867,Z 80,A 157.4284,B 24.8923,C -2.3951,E1 24.8467,E2 -73.0227} C_DIS
LIN {X -68.186,Y 23.4933,Z 80,A 154.5447,B 24.8916,C -2.4029,E1 24.8492,E2 -70.1411} C_DIS
LIN {X -67.146,Y 26.3159,Z 80,A 152.3074,B 24.8907,C -2.4135,E1 24.8515,E2 -67.9165} C_DIS
LIN {X -65.9341,Y 29.2218,Z 80,A 149.6637,B 24.8903,C -2.4178,E1 24.8544,E2 -65.2685} C_DIS
LIN {X -64.4298,Y 32.4035,Z 80,A 146.9968,B 24.8893,C -2.4289,E1 24.8576,E2 -62.6137} C_DIS
LIN {X -63.1837,Y 34.7719,Z 80,A 144.7491,B 24.889,C -2.4324,E1 24.8606,E2 -60.3623} C_DIS
LIN {X -61.5655,Y 37.5607,Z 80,A 142.3686,B 24.8879,C -2.4436,E1 24.864,E2 -57.9964} C_DIS
LIN {X -59.9522,Y 40.087,Z 80,A 139.8475,B 24.8876,C -2.4471,E1 24.8678,E2 -55.4709} C_DIS
LIN {X -58.2323,Y 42.5455,Z 80,A 137.5033,B 24.8869,C -2.4544,E1 24.8716,E2 -53.1327} C_DIS
LIN {X -56.4196,Y 44.922,Z 80,A 134.9847,B 24.8867,C -2.4574,E1 24.8759,E2 -50.6094} C_DIS
LIN {X -54.3208,Y 47.4379,Z 80,A 132.3246,B 24.8862,C -2.4628,E1 24.8808,E2 -47.95} C_DIS
LIN {X -52.0265,Y 49.9437,Z 80,A 129.766,B 24.8853,C -2.4726,E1 24.8856,E2 -45.4035} C_DIS
LIN {X -49.9095,Y 52.0595,Z 80,A 127.2884,B 24.8849,C -2.4759,E1 24.8906,E2 -42.9235} C_DIS
LIN {X -47.5622,Y 54.2123,Z 80,A 124.7968,B 24.8843,C -2.4825,E1 24.8957,E2 -40.4377} C_DIS
LIN {X -45.0479,Y 56.3198,Z 80,A 122.1451,B 24.8839,C -2.4871,E1 24.9014,E2 -37.787} C_DIS
LIN {X -42.9562,Y 57.9312,Z 80,A 120.1038,B 24.8834,C -2.4928,E1 24.906,E2 -35.7517} C_DIS
LIN {X -40.7991,Y 59.4695,Z 80,A 117.9333,B 24.8831,C -2.4954,E1 24.911,E2 -33.5801} C_DIS
LIN {X -38.572,Y 60.9384,Z 80,A 115.8397,B 24.8827,C -2.5,E1 24.9159,E2 -31.4907} C_DIS
LIN {X -36.145,Y 62.4076,Z 80,A 113.4957,B 24.8825,C -2.5019,E1 24.9215,E2 -29.1443} C_DIS
LIN {X -33.4867,Y 63.8725,Z 80,A 111.272,B 24.8817,C -2.5104,E1 24.9269,E2 -26.9344} C_DIS
LIN {X -30.8272,Y 65.1987,Z 80,A 108.6587,B 24.8819,C -2.5081,E1 24.9335,E2 -24.309} C_DIS
LIN {X -27.5872,Y 66.6332,Z 80,A 105.9956,B 24.8812,C -2.5158,E1 24.9403,E2 -21.6579} C_DIS
LIN {X -24.7703,Y 67.7314,Z 80,A 103.6151,B 24.8809,C -2.5194,E1 24.9465,E2 -19.281} C_DIS
LIN {X -21.6917,Y 68.78,Z 80,A 100.8487,B 24.8809,C -2.5181,E1 24.9539,E2 -16.5064} C_DIS
LIN {X -18.3421,Y 69.748,Z 80,A 98.0341,B 24.8809,C -2.5199,E1 24.9615,E2 -13.6917} C_DIS
LIN {X -15.4217,Y 70.4506,Z 80,A 95.671,B 24.8805,C -2.5226,E1 24.9679,E2 -11.332} C_DIS
LIN {X -12.3368,Y 71.0566,Z 80,A 93.323,B 24.88,C -2.5281,E1 24.9743,E2 -8.9947} C_DIS
LIN {X -9.7325,Y 71.4598,Z 80,A 91.106,B 24.8802,C -2.5265,E1 24.9804,E2 -6.7719} C_DIS
LIN {X -6.5579,Y 71.82,Z 80,A 88.5791,B 24.88,C -2.5281,E1 24.9875,E2 -4.2473} C_DIS
LIN {X -3.5279,Y 72.033,Z 80,A 86.0895,B 24.8801,C -2.5271,E1 24.9944,E2 -1.7547} C_DIS
LIN {X -0.3673,Y 72.1178,Z 80,A 83.6501,B 24.8799,C -2.5295,E1 25.0012,E2 0.6792} C_DIS
LIN {X 2.7065,Y 72.0675,Z 80,A 81.3611,B 24.8795,C -2.5336,E1 25.0076,E2 2.958} C_DIS
LIN {X 5.3272,Y 71.9214,Z 80,A 79.2789,B 24.8795,C -2.5336,E1 25.0134,E2 5.0391} C_DIS
LIN {X 7.9492,Y 71.6791,Z 80,A 77.1063,B 24.8797,C -2.5314,E1 25.0194,E2 7.2158} C_DIS
LIN {X 10.6269,Y 71.3326,Z 80,A 74.9805,B 24.8797,C -2.5314,E1 25.0253,E2 9.3398} C_DIS
LIN {X 13.2236,Y 70.8967,Z 80,A 72.7451,B 24.8801,C -2.5269,E1 25.0314,E2 11.5833} C_DIS
LIN {X 16.1939,Y 70.2771,Z 80,A 70.4721,B 24.8799,C -2.5293,E1 25.0376,E2 13.8477} C_DIS
LIN {X 18.7332,Y 69.6432,Z 80,A 68.4357,B 24.8799,C -2.5291,E1 25.0431,E2 15.8814} C_DIS
LIN {X 21.7823,Y 68.7519,Z 80,A 65.7371,B 24.8805,C -2.5227,E1 25.0504,E2 18.5904} C_DIS
LIN {X 25.1299,Y 67.5982,Z 80,A 63.148,B 24.8802,C -2.5261,E1 25.0571,E2 21.1662} C_DIS
LIN {X 27.5978,Y 66.6288,Z 80,A 60.8676,B 24.8808,C -2.5194,E1 25.0631,E2 23.4572} C_DIS
LIN {X 30.7918,Y 65.2154,Z 80,A 58.1937,B 24.8808,C -2.5189,E1 25.0698,E2 26.1256} C_DIS
LIN {X 33.2293,Y 64.0074,Z 80,A 56.0403,B 24.8811,C -2.5164,E1 25.0752,E2 28.2791} C_DIS
LIN {X 35.5579,Y 62.7449,Z 80,A 53.951,B 24.8814,C -2.5139,E1 25.0803,E2 30.3682} C_DIS
LIN {X 37.837,Y 61.3972,Z 80,A 51.814,B 24.8817,C -2.5099,E1 25.0854,E2 32.508} C_DIS
LIN {X 40.3742,Y 59.7582,Z 80,A 49.4653,B 24.882,C -2.5075,E1 25.0909,E2 34.8546} C_DIS
LIN {X 42.5636,Y 58.2189,Z 80,A 47.3768,B 24.8822,C -2.5049,E1 25.0956,E2 36.9419} C_DIS
LIN {X 44.9182,Y 56.4226,Z 80,A 44.884,B 24.883,C -2.4969,E1 25.1011,E2 39.4445} C_DIS
LIN {X 47.4442,Y 54.3154,Z 80,A 42.334,B 24.8833,C -2.4937,E1 25.1066,E2 41.9923} C_DIS
LIN {X 49.7301,Y 52.2312,Z 80,A 39.9341,B 24.8836,C -2.4903,E1 25.1115,E2 44.3904} C_DIS
LIN {X 51.8198,Y 50.1582,Z 80,A 37.6175,B 24.884,C -2.4859,E1 25.116,E2 46.7074} C_DIS
LIN {X 54.0349,Y 47.7643,Z 80,A 34.9259,B 24.8848,C -2.4774,E1 25.1211,E2 49.4072} C_DIS
LIN {X 56.3006,Y 45.0721,Z 80,A 32.1834,B 24.8853,C -2.4724,E1 25.1259,E2 52.1489} C_DIS
LIN {X 58.2332,Y 42.5441,Z 80,A 29.6602,B 24.8858,C -2.4664,E1 25.1302,E2 54.6742} C_DIS
LIN {X 59.9641,Y 40.0692,Z 80,A 27.2335,B 24.8865,C -2.4596,E1 25.134,E2 57.105} C_DIS
LIN {X 61.5882,Y 37.5235,Z 80,A 25.0235,B 24.8865,C -2.4587,E1 25.1372,E2 59.3059} C_DIS
LIN {X 62.9235,Y 35.2384,Z 80,A 22.8994,B 24.8871,C -2.4525,E1 25.1402,E2 61.4337} C_DIS
LIN {X 64.253,Y 32.7516,Z 80,A 20.7054,B 24.8876,C -2.4477,E1 25.143,E2 63.6274} C_DIS
LIN {X 65.4127,Y 30.3686,Z 80,A 18.659,B 24.8879,C -2.4435,E1 25.1455,E2 65.6727} C_DIS
LIN {X 66.6279,Y 27.5999,Z 80,A 16.1954,B 24.8887,C -2.435,E1 25.1482,E2 68.143} C_DIS
LIN {X 67.7295,Y 24.7754,Z 80,A 13.8094,B 24.8893,C -2.4286,E1 25.1506,E2 70.5308} C_DIS
LIN {X 68.759,Y 21.7593,Z 80,A 11.1346,B 24.8904,C -2.4171,E1 25.1529,E2 73.2177} C_DIS
LIN {X 69.7365,Y 18.3866,Z 80,A 8.3115,B 24.8912,C -2.4078,E1 25.155,E2 76.0465} C_DIS
LIN {X 70.5671,Y 14.8823,Z 80,A 5.6382,B 24.8915,C -2.4044,E1 25.1567,E2 78.7124} C_DIS
LIN {X 71.073,Y 12.2415,Z 80,A 3.5647,B 24.8919,C -2.3996,E1 25.1577,E2 80.7851} C_DIS
LIN {X 71.4646,Y 9.6962,Z 80,A 1.4786,B 24.8926,C -2.392,E1 25.1585,E2 82.8767} C_DIS
LIN {X 71.7713,Y 7.0659,Z 80,A -0.5228,B 24.893,C -2.3884,E1 25.1591,E2 84.8749} C_DIS
LIN {X 71.9965,Y 4.2019,Z 80,A -2.9333,B 24.8939,C -2.3775,E1 25.1596,E2 87.2967} C_DIS
LIN {X 72.1076,Y 1.2655,Z 80,A -5.2302,B 24.8945,C -2.3712,E1 25.1598,E2 89.595} C_DIS
LIN {X 72.0968,Y -1.7724,Z 80,A -7.5614,B 24.895,C -2.3659,E1 25.1597,E2 91.9248} C_DIS
LIN {X 71.9831,Y -4.4213,Z 80,A -9.771,B 24.8958,C -2.3562,E1 25.1594,E2 94.1441} C_DIS
LIN {X 71.6797,Y -7.9431,Z 80,A -12.2412,B 24.8958,C -2.357,E1 25.1587,E2 96.5979} C_DIS
LIN {X 71.3191,Y -10.7142,Z 80,A -14.5954,B 24.8967,C -2.346,E1 25.1578,E2 98.9641} C_DIS
LIN {X 70.8966,Y -13.224,Z 80,A -16.7991,B 24.8977,C -2.3344,E1 25.1567,E2 101.1823} C_DIS
LIN {X 70.2807,Y -16.1782,Z 80,A -19.0544,B 24.8981,C -2.331,E1 25.1554,E2 103.4326} C_DIS
LIN {X 69.64,Y -18.7453,Z 80,A -21.1131,B 24.8985,C -2.3256,E1 25.1539,E2 105.4922} C_DIS
LIN {X 68.7543,Y -21.7747,Z 80,A -23.756,B 24.8995,C -2.3139,E1 25.1518,E2 108.1475} C_DIS
LIN {X 67.6046,Y -25.1127,Z 80,A -26.335,B 24.8997,C -2.3118,E1 25.1494,E2 110.7171} C_DIS
LIN {X 66.6304,Y -27.594,Z 80,A -28.6135,B 24.9007,C -2.3008,E1 25.147,E2 113.009} C_DIS
LIN {X 65.3618,Y -30.4787,Z 80,A -30.9836,B 24.901,C -2.2971,E1 25.1443,E2 115.375} C_DIS
LIN {X 64.1606,Y -32.9325,Z 80,A -33.2766,B 24.9019,C -2.2872,E1 25.1414,E2 117.6791} C_DIS
Enddeposition()
END
